LIN {X 0,Y 199.648,Z 315.611,A -85,B 0,C 180,E1 -21577.217,E2 -21577.217} C_VEL
LIN {X 0,Y 199.715,Z 315.609,A -85,B 0,C 180,E1 -21581.799,E2 -21581.799} C_VEL
LIN {X 0,Y 199.766,Z 315.596,A -85,B 0,C 180,E1 -21585.742,E2 -21585.742} C_VEL
LIN {X 0,Y 199.991,Z 315.572,A -85,B 0,C 180,E1 -21589.879,E2 -21589.879} C_VEL
LIN {X 0,Y 199.982,Z 315.569,A -85,B 0,C 180,E1 -21593.947,E2 -21593.947} C_VEL
LIN {X 0,Y 200.285,Z 315.535,A -85,B 0,C 180,E1 -21597.988,E2 -21597.988} C_VEL
LIN {X 0,Y 200.436,Z 315.515,A -85,B 0,C 180,E1 -21599.999,E2 -21599.999} C_VEL
LIN {X 0,Y 199.983,Z 315.57,A -85,B 0,C 180,E1 -21604.029,E2 -21604.029} C_VEL
LIN {X 0,Y 200.046,Z 315.564,A -85,B 0,C 180,E1 -21608.077,E2 -21608.077} C_VEL
LIN {X 0,Y 199.831,Z 315.588,A -85,B 0,C 180,E1 -21612.181,E2 -21612.181} C_VEL
LIN {X 0,Y 199.759,Z 315.601,A -85,B 0,C 180,E1 -21616.346,E2 -21616.346} C_VEL
LIN {X 0,Y 199.644,Z 315.611,A -85,B 0,C 180,E1 -21620.61,E2 -21620.61} C_VEL
LIN {X 0,Y 199.625,Z 315.617,A -85,B 0,C 180,E1 -21624.99,E2 -21624.99} C_VEL
LIN {X 0,Y 199.594,Z 315.616,A -85,B 0,C 180,E1 -21629.534,E2 -21629.534} C_VEL
LIN {X 0,Y 199.635,Z 315.616,A -85,B 0,C 180,E1 -21632.355,E2 -21632.355} C_VEL
LIN {X 0,Y 199.59,Z 315.623,A -85,B 0,C 180,E1 -21636.769,E2 -21636.769} C_VEL
LIN {X 0,Y 199.569,Z 315.628,A -85,B 0,C 180,E1 -21639.336,E2 -21639.336} C_VEL
LIN {X 0,Y 199.544,Z 315.627,A -85,B 0,C 180,E1 -21642.313,E2 -21642.313} C_VEL
LIN {X 0,Y 199.554,Z 315.629,A -85,B 0,C 180,E1 -21645.233,E2 -21645.233} C_VEL
LIN {X 0,Y 199.69,Z 315.812,A -85,B 0,C 180,E1 -21650.538,E2 -21650.538} C_VEL
LIN {X 0,Y 202.068,Z 326.672,A -85,B 0,C 180,E1 -21654.989,E2 -21654.989} C_VEL
LIN {X 0,Y 204.574,Z 338.295,A -85,B 0,C 180,E1 -21659.506,E2 -21659.506} C_VEL
LIN {X 0,Y 205.421,Z 343.365,A -85,B 0,C 180,E1 -21661.389,E2 -21661.389} C_VEL
LIN {X 0,Y 205.397,Z 343.737,A -85,B 0,C 180,E1 -21661.521,E2 -21661.521} C_VEL
LIN {X 0,Y 206.412,Z 366.002,A -85,B 0,C 180,E1 -21662.678,E2 -21662.678} C_VEL
LIN {X 0,Y 207.666,Z 381.182,A -85,B 0,C 180,E1 -21663.491,E2 -21663.491} C_VEL
LIN {X 0,Y 207.515,Z 385.039,A -85,B 0,C 180,E1 -21663.67,E2 -21663.67} C_VEL
LIN {X 0,Y 206.711,Z 388.85,A -85,B 0,C 180,E1 -21663.813,E2 -21663.813} C_VEL
LIN {X 0,Y 200.517,Z 405.605,A -85,B 0,C 180,E1 -21664.357,E2 -21664.357} C_VEL
LIN {X 0,Y 199.538,Z 411.412,A -85,B 0,C 180,E1 -21664.613,E2 -21664.613} C_VEL
LIN {X 0,Y 198.167,Z 444.281,A -85,B 0,C 180,E1 -21666.285,E2 -21666.285} C_VEL
LIN {X 0,Y 197.452,Z 454.911,A -85,B 0,C 180,E1 -21667.096,E2 -21667.096} C_VEL
LIN {X 0,Y 196.39,Z 466.849,A -85,B 0,C 180,E1 -21668.351,E2 -21668.351} C_VEL
LIN {X 0,Y 195.216,Z 478.665,A -85,B 0,C 180,E1 -21670.039,E2 -21670.039} C_VEL
LIN {X 0,Y 194.149,Z 488.366,A -85,B 0,C 180,E1 -21671.813,E2 -21671.813} C_VEL
LIN {X 0,Y 193.082,Z 497.591,A -85,B 0,C 180,E1 -21673.892,E2 -21673.892} C_VEL
LIN {X 0,Y 192.324,Z 504.426,A -85,B 0,C 180,E1 -21675.726,E2 -21675.726} C_VEL
LIN {X 0,Y 191.715,Z 511.1,A -85,B 0,C 180,E1 -21677.837,E2 -21677.837} C_VEL
LIN {X 0,Y 191.271,Z 518.01,A -85,B 0,C 180,E1 -21680.488,E2 -21680.488} C_VEL
LIN {X 0,Y 191.048,Z 523.997,A -85,B 0,C 180,E1 -21683.323,E2 -21683.323} C_VEL
LIN {X 0,Y 190.99,Z 528.22,A -85,B 0,C 180,E1 -21685.784,E2 -21685.784} C_VEL
LIN {X 0,Y 190.988,Z 532.388,A -85,B 0,C 180,E1 -21688.95,E2 -21688.95} C_VEL
LIN {X 0,Y 191.131,Z 533.502,A -85,B 0,C 180,E1 -21690.004,E2 -21690.004} C_VEL
LIN {X 0,Y 190.578,Z 536.736,A -85,B 0,C 180,E1 -21694.234,E2 -21694.234} C_VEL
LIN {X 0,Y 190.558,Z 538.115,A -85,B 0,C 180,E1 -21698.487,E2 -21698.487} C_VEL
LIN {X 0,Y 190.933,Z 538.228,A -85,B 0,C 180,E1 -21700.609,E2 -21700.609} C_VEL
LIN {X 0,Y 192.399,Z 537.275,A -85,B 0,C 180,E1 -21704.818,E2 -21704.818} C_VEL
LIN {X 0,Y 195.192,Z 534.63,A -85,B 0,C 180,E1 -21708.91,E2 -21708.91} C_VEL
LIN {X 0,Y 197.896,Z 531.626,A -85,B 0,C 180,E1 -21711.896,E2 -21711.896} C_VEL
LIN {X 0,Y 201.136,Z 527.628,A -85,B 0,C 180,E1 -21714.792,E2 -21714.792} C_VEL
LIN {X 0,Y 205.16,Z 522.48,A -85,B 0,C 180,E1 -21717.547,E2 -21717.547} C_VEL
LIN {X 0,Y 208.994,Z 517.234,A -85,B 0,C 180,E1 -21719.738,E2 -21719.738} C_VEL
LIN {X 0,Y 213.102,Z 511.034,A -85,B 0,C 180,E1 -21721.849,E2 -21721.849} C_VEL
LIN {X 0,Y 216.699,Z 505.229,A -85,B 0,C 180,E1 -21723.46,E2 -21723.46} C_VEL
LIN {X 0,Y 221.524,Z 496.519,A -85,B 0,C 180,E1 -21725.38,E2 -21725.38} C_VEL
LIN {X 0,Y 225.582,Z 488.226,A -85,B 0,C 180,E1 -21726.851,E2 -21726.851} C_VEL
LIN {X 0,Y 229.297,Z 479.732,A -85,B 0,C 180,E1 -21728.085,E2 -21728.085} C_VEL
LIN {X 0,Y 232.642,Z 471.031,A -85,B 0,C 180,E1 -21729.096,E2 -21729.096} C_VEL
LIN {X 0,Y 236.162,Z 460.215,A -85,B 0,C 180,E1 -21730.056,E2 -21730.056} C_VEL
LIN {X 0,Y 238.892,Z 449.846,A -85,B 0,C 180,E1 -21730.748,E2 -21730.748} C_VEL
LIN {X 0,Y 241.019,Z 439.165,A -85,B 0,C 180,E1 -21731.279,E2 -21731.279} C_VEL
LIN {X 0,Y 246.635,Z 399.578,A -85,B 0,C 180,E1 -21732.928,E2 -21732.928} C_VEL
LIN {X 0,Y 244.463,Z 393.666,A -85,B 0,C 180,E1 -21734.894,E2 -21734.894} C_VEL
LIN {X 0,Y 242.901,Z 389.862,A -85,B 0,C 180,E1 -21736.566,E2 -21736.566} C_VEL
LIN {X 0,Y 241.28,Z 386.207,A -85,B 0,C 180,E1 -21738.592,E2 -21738.592} C_VEL
LIN {X 0,Y 239.343,Z 382.083,A -85,B 0,C 180,E1 -21742.091,E2 -21742.091} C_VEL
LIN {X 0,Y 238.603,Z 380.779,A -85,B 0,C 180,E1 -21744.45,E2 -21744.45} C_VEL
LIN {X 0,Y 238.575,Z 380.682,A -85,B 0,C 180,E1 -21748.678,E2 -21748.678} C_VEL
LIN {X 0,Y 239.448,Z 381.752,A -85,B 0,C 180,E1 -21751.296,E2 -21751.296} C_VEL
LIN {X 0,Y 241.721,Z 386.414,A -85,B 0,C 180,E1 -21755.249,E2 -21755.249} C_VEL
LIN {X 0,Y 243.812,Z 390.848,A -85,B 0,C 180,E1 -21757.643,E2 -21757.643} C_VEL
LIN {X 0,Y 245.743,Z 395.641,A -85,B 0,C 180,E1 -21759.539,E2 -21759.539} C_VEL
LIN {X 0,Y 246.432,Z 397.591,A -85,B 0,C 180,E1 -21760.175,E2 -21760.175} C_VEL
LIN {X 0,Y 240.499,Z 435.091,A -85,B 0,C 180,E1 -21761.871,E2 -21761.871} C_VEL
LIN {X 0,Y 237.483,Z 448.761,A -85,B 0,C 180,E1 -21762.787,E2 -21762.787} C_VEL
LIN {X 0,Y 234.505,Z 458.837,A -85,B 0,C 180,E1 -21763.725,E2 -21763.725} C_VEL
LIN {X 0,Y 231.305,Z 467.899,A -85,B 0,C 180,E1 -21764.808,E2 -21764.808} C_VEL
LIN {X 0,Y 227.57,Z 476.863,A -85,B 0,C 180,E1 -21766.153,E2 -21766.153} C_VEL
LIN {X 0,Y 223.672,Z 484.895,A -85,B 0,C 180,E1 -21767.65,E2 -21767.65} C_VEL
LIN {X 0,Y 219.496,Z 492.508,A -85,B 0,C 180,E1 -21769.392,E2 -21769.392} C_VEL
LIN {X 0,Y 214.975,Z 499.839,A -85,B 0,C 180,E1 -21771.541,E2 -21771.541} C_VEL
LIN {X 0,Y 209.923,Z 506.722,A -85,B 0,C 180,E1 -21774.237,E2 -21774.237} C_VEL
LIN {X 0,Y 205.514,Z 511.853,A -85,B 0,C 180,E1 -21776.975,E2 -21776.975} C_VEL
LIN {X 0,Y 202.853,Z 514.621,A -85,B 0,C 180,E1 -21778.909,E2 -21778.909} C_VEL
LIN {X 0,Y 199.2,Z 517.68,A -85,B 0,C 180,E1 -21782.023,E2 -21782.023} C_VEL
LIN {X 0,Y 197.206,Z 519.017,A -85,B 0,C 180,E1 -21784.088,E2 -21784.088} C_VEL
LIN {X 0,Y 195.451,Z 519.821,A -85,B 0,C 180,E1 -21786.194,E2 -21786.194} C_VEL
LIN {X 0,Y 193.934,Z 520.014,A -85,B 0,C 180,E1 -21788.336,E2 -21788.336} C_VEL
LIN {X 0,Y 192.716,Z 519.734,A -85,B 0,C 180,E1 -21790.507,E2 -21790.507} C_VEL
LIN {X 0,Y 191.73,Z 518.983,A -85,B 0,C 180,E1 -21792.706,E2 -21792.706} C_VEL
LIN {X 0,Y 190.999,Z 517.686,A -85,B 0,C 180,E1 -21794.927,E2 -21794.927} C_VEL
LIN {X 0,Y 190.342,Z 514.593,A -85,B 0,C 180,E1 -21798.292,E2 -21798.292} C_VEL
LIN {X 0,Y 190.255,Z 511.807,A -85,B 0,C 180,E1 -21800.545,E2 -21800.545} C_VEL
LIN {X 0,Y 190.441,Z 506.225,A -85,B 0,C 180,E1 -21803.951,E2 -21803.951} C_VEL
LIN {X 0,Y 190.888,Z 500.472,A -85,B 0,C 180,E1 -21806.689,E2 -21806.689} C_VEL
LIN {X 0,Y 191.39,Z 494.218,A -85,B 0,C 180,E1 -21809.115,E2 -21809.115} C_VEL
LIN {X 0,Y 191.861,Z 488.925,A -85,B 0,C 180,E1 -21810.854,E2 -21810.854} C_VEL
LIN {X 0,Y 192.742,Z 480.468,A -85,B 0,C 180,E1 -21813.159,E2 -21813.159} C_VEL
LIN {X 0,Y 193.68,Z 471.435,A -85,B 0,C 180,E1 -21815.175,E2 -21815.175} C_VEL
LIN {X 0,Y 194.762,Z 460.212,A -85,B 0,C 180,E1 -21817.189,E2 -21817.189} C_VEL
LIN {X 0,Y 195.736,Z 448.504,A -85,B 0,C 180,E1 -21818.765,E2 -21818.765} C_VEL
LIN {X 0,Y 196.492,Z 438.184,A -85,B 0,C 180,E1 -21819.827,E2 -21819.827} C_VEL
LIN {X 0,Y 197.164,Z 426.158,A -85,B 0,C 180,E1 -21820.726,E2 -21820.726} C_VEL
LIN {X 0,Y 199.44,Z 377.415,A -85,B 0,C 180,E1 -21823.388,E2 -21823.388} C_VEL
LIN {X 0,Y 196.403,Z 343.515,A -85,B 0,C 180,E1 -21825.476,E2 -21825.476} C_VEL
LIN {X 0,Y 196.313,Z 340.974,A -85,B 0,C 180,E1 -21825.635,E2 -21825.635} C_VEL
LIN {X 0,Y 196.727,Z 336.975,A -85,B 0,C 180,E1 -21827.252,E2 -21827.252} C_VEL
LIN {X 0,Y 194.607,Z 325.863,A -85,B 0,C 180,E1 -21832.125,E2 -21832.125} C_VEL
LIN {X 0,Y 192.67,Z 316.483,A -85,B 0,C 180,E1 -21836.514,E2 -21836.514} C_VEL
LIN {X 0,Y 192.616,Z 316.492,A -85,B 0,C 180,E1 -21841.682,E2 -21841.682} C_VEL
LIN {X 0,Y 192.662,Z 316.489,A -85,B 0,C 180,E1 -21846.341,E2 -21846.341} C_VEL
LIN {X 0,Y 192.701,Z 316.479,A -85,B 0,C 180,E1 -21851.49,E2 -21851.49} C_VEL
LIN {X 0,Y 192.735,Z 316.472,A -85,B 0,C 180,E1 -21855.209,E2 -21855.209} C_VEL
LIN {X 0,Y 192.952,Z 316.449,A -85,B 0,C 180,E1 -21859.564,E2 -21859.564} C_VEL
LIN {X 0,Y 192.968,Z 316.444,A -85,B 0,C 180,E1 -21863.724,E2 -21863.724} C_VEL
LIN {X 0,Y 193.231,Z 316.415,A -85,B 0,C 180,E1 -21867.912,E2 -21867.912} C_VEL
LIN {X 0,Y 193.417,Z 316.392,A -85,B 0,C 180,E1 -21869.996,E2 -21869.996} C_VEL
LIN {X 0,Y 192.934,Z 316.449,A -85,B 0,C 180,E1 -21874.173,E2 -21874.173} C_VEL
LIN {X 0,Y 193.028,Z 316.441,A -85,B 0,C 180,E1 -21878.369,E2 -21878.369} C_VEL
LIN {X 0,Y 192.794,Z 316.466,A -85,B 0,C 180,E1 -21882.628,E2 -21882.628} C_VEL
LIN {X 0,Y 192.715,Z 316.48,A -85,B 0,C 180,E1 -21886.956,E2 -21886.956} C_VEL
LIN {X 0,Y 192.578,Z 316.491,A -85,B 0,C 180,E1 -21891.397,E2 -21891.397} C_VEL
LIN {X 0,Y 192.63,Z 316.487,A -85,B 0,C 180,E1 -21894.198,E2 -21894.198} C_VEL
LIN {X 0,Y 192.593,Z 316.492,A -85,B 0,C 180,E1 -21898.858,E2 -21898.858} C_VEL
LIN {X 0,Y 192.584,Z 316.493,A -85,B 0,C 180,E1 -21903.18,E2 -21903.18} C_VEL
LIN {X 0,Y 192.528,Z 316.498,A -85,B 0,C 180,E1 -21908.347,E2 -21908.347} C_VEL
LIN {X 0,Y 192.471,Z 316.508,A -85,B 0,C 180,E1 -21913.087,E2 -21913.087} C_VEL
LIN {X 0,Y 192.468,Z 316.506,A -85,B 0,C 180,E1 -21916.9,E2 -21916.9} C_VEL
LIN {X 0,Y 192.52,Z 316.501,A -85,B 0,C 180,E1 -21921.639,E2 -21921.639} C_VEL
LIN {X 0,Y 192.572,Z 316.494,A -85,B 0,C 180,E1 -21926.808,E2 -21926.808} C_VEL
LIN {X 0,Y 192.638,Z 316.488,A -85,B 0,C 180,E1 -21931.686,E2 -21931.686} C_VEL
LIN {X 0,Y 192.644,Z 316.482,A -85,B 0,C 180,E1 -21936.339,E2 -21936.339} C_VEL
LIN {X 0,Y 192.664,Z 316.486,A -85,B 0,C 180,E1 -21941.488,E2 -21941.488} C_VEL
LIN {X 0,Y 192.692,Z 316.475,A -85,B 0,C 180,E1 -21945.207,E2 -21945.207} C_VEL
LIN {X 0,Y 192.914,Z 316.453,A -85,B 0,C 180,E1 -21949.564,E2 -21949.564} C_VEL
LIN {X 0,Y 192.944,Z 316.445,A -85,B 0,C 180,E1 -21953.725,E2 -21953.725} C_VEL
LIN {X 0,Y 193.227,Z 316.414,A -85,B 0,C 180,E1 -21957.914,E2 -21957.914} C_VEL
LIN {X 0,Y 193.401,Z 316.392,A -85,B 0,C 180,E1 -21959.999,E2 -21959.999} C_VEL
LIN {X 0,Y 192.929,Z 316.448,A -85,B 0,C 180,E1 -21964.177,E2 -21964.177} C_VEL
LIN {X 0,Y 192.996,Z 316.442,A -85,B 0,C 180,E1 -21968.374,E2 -21968.374} C_VEL
LIN {X 0,Y 192.759,Z 316.469,A -85,B 0,C 180,E1 -21972.635,E2 -21972.635} C_VEL
LIN {X 0,Y 192.717,Z 316.477,A -85,B 0,C 180,E1 -21976.961,E2 -21976.961} C_VEL
LIN {X 0,Y 192.578,Z 316.491,A -85,B 0,C 180,E1 -21981.403,E2 -21981.403} C_VEL
LIN {X 0,Y 192.61,Z 316.493,A -85,B 0,C 180,E1 -21984.211,E2 -21984.211} C_VEL
LIN {X 0,Y 192.592,Z 316.489,A -85,B 0,C 180,E1 -21988.88,E2 -21988.88} C_VEL
LIN {X 0,Y 192.566,Z 316.498,A -85,B 0,C 180,E1 -21993.191,E2 -21993.191} C_VEL
LIN {X 0,Y 192.516,Z 316.504,A -85,B 0,C 180,E1 -21998.359,E2 -21998.359} C_VEL
LIN {X 0,Y 192.463,Z 316.512,A -85,B 0,C 180,E1 -22003.099,E2 -22003.099} C_VEL
LIN {X 0,Y 192.467,Z 316.51,A -85,B 0,C 180,E1 -22006.911,E2 -22006.911} C_VEL
LIN {X 0,Y 192.604,Z 316.676,A -85,B 0,C 180,E1 -22010.019,E2 -22010.019} C_VEL
LIN {X 0,Y 194.779,Z 326.353,A -85,B 0,C 180,E1 -22014.143,E2 -22014.143} C_VEL
LIN {X 0,Y 197.226,Z 337.828,A -85,B 0,C 180,E1 -22018.782,E2 -22018.782} C_VEL
LIN {X 0,Y 198.356,Z 343.639,A -85,B 0,C 180,E1 -22021.049,E2 -22021.049} C_VEL
LIN {X 0,Y 199.807,Z 370.761,A -85,B 0,C 180,E1 -22022.547,E2 -22022.547} C_VEL
LIN {X 0,Y 200.674,Z 384.052,A -85,B 0,C 180,E1 -22023.276,E2 -22023.276} C_VEL
LIN {X 0,Y 199.538,Z 411.412,A -85,B 0,C 180,E1 -22024.613,E2 -22024.613} C_VEL
LIN {X 0,Y 198.65,Z 417.188,A -85,B 0,C 180,E1 -22024.865,E2 -22024.865} C_VEL
LIN {X 0,Y 192.214,Z 435.809,A -85,B 0,C 180,E1 -22025.563,E2 -22025.563} C_VEL
LIN {X 0,Y 191.277,Z 441.55,A -85,B 0,C 180,E1 -22025.881,E2 -22025.881} C_VEL
LIN {X 0,Y 190.616,Z 452.157,A -85,B 0,C 180,E1 -22026.657,E2 -22026.657} C_VEL
LIN {X 0,Y 189.733,Z 462.427,A -85,B 0,C 180,E1 -22027.695,E2 -22027.695} C_VEL
LIN {X 0,Y 188.828,Z 471.698,A -85,B 0,C 180,E1 -22028.901,E2 -22028.901} C_VEL
LIN {X 0,Y 187.89,Z 480.588,A -85,B 0,C 180,E1 -22030.334,E2 -22030.334} C_VEL
LIN {X 0,Y 186.975,Z 488.81,A -85,B 0,C 180,E1 -22031.941,E2 -22031.941} C_VEL
LIN {X 0,Y 186.029,Z 496.842,A -85,B 0,C 180,E1 -22033.828,E2 -22033.828} C_VEL
LIN {X 0,Y 185.277,Z 503.711,A -85,B 0,C 180,E1 -22035.732,E2 -22035.732} C_VEL
LIN {X 0,Y 184.574,Z 511.846,A -85,B 0,C 180,E1 -22038.474,E2 -22038.474} C_VEL
LIN {X 0,Y 184.224,Z 517.336,A -85,B 0,C 180,E1 -22040.675,E2 -22040.675} C_VEL
LIN {X 0,Y 184.043,Z 523.013,A -85,B 0,C 180,E1 -22043.427,E2 -22043.427} C_VEL
LIN {X 0,Y 183.993,Z 526.802,A -85,B 0,C 180,E1 -22045.624,E2 -22045.624} C_VEL
LIN {X 0,Y 183.975,Z 531.244,A -85,B 0,C 180,E1 -22048.91,E2 -22048.91} C_VEL
LIN {X 0,Y 184.118,Z 532.372,A -85,B 0,C 180,E1 -22050.004,E2 -22050.004} C_VEL
LIN {X 0,Y 183.695,Z 534.391,A -85,B 0,C 180,E1 -22052.197,E2 -22052.197} C_VEL
LIN {X 0,Y 183.455,Z 536.25,A -85,B 0,C 180,E1 -22055.117,E2 -22055.117} C_VEL
LIN {X 0,Y 183.535,Z 537.535,A -85,B 0,C 180,E1 -22058.814,E2 -22058.814} C_VEL
LIN {X 0,Y 184.599,Z 537.553,A -85,B 0,C 180,E1 -22063.208,E2 -22063.208} C_VEL
LIN {X 0,Y 185.515,Z 537.031,A -85,B 0,C 180,E1 -22065.381,E2 -22065.381} C_VEL
LIN {X 0,Y 188.465,Z 534.759,A -85,B 0,C 180,E1 -22069.613,E2 -22069.613} C_VEL
LIN {X 0,Y 191.326,Z 531.999,A -85,B 0,C 180,E1 -22072.689,E2 -22072.689} C_VEL
LIN {X 0,Y 194.746,Z 528.239,A -85,B 0,C 180,E1 -22075.664,E2 -22075.664} C_VEL
LIN {X 0,Y 198.959,Z 523.417,A -85,B 0,C 180,E1 -22078.483,E2 -22078.483} C_VEL
LIN {X 0,Y 203.777,Z 517.353,A -85,B 0,C 180,E1 -22081.155,E2 -22081.155} C_VEL
LIN {X 0,Y 208.14,Z 511.24,A -85,B 0,C 180,E1 -22083.278,E2 -22083.278} C_VEL
LIN {X 0,Y 212.908,Z 503.926,A -85,B 0,C 180,E1 -22085.287,E2 -22085.287} C_VEL
LIN {X 0,Y 216.99,Z 497.107,A -85,B 0,C 180,E1 -22086.812,E2 -22086.812} C_VEL
LIN {X 0,Y 221.791,Z 487.937,A -85,B 0,C 180,E1 -22088.453,E2 -22088.453} C_VEL
LIN {X 0,Y 225.676,Z 479.438,A -85,B 0,C 180,E1 -22089.673,E2 -22089.673} C_VEL
LIN {X 0,Y 229.172,Z 470.724,A -85,B 0,C 180,E1 -22090.667,E2 -22090.667} C_VEL
LIN {X 0,Y 232.839,Z 460.044,A -85,B 0,C 180,E1 -22091.609,E2 -22091.609} C_VEL
LIN {X 0,Y 235.699,Z 449.867,A -85,B 0,C 180,E1 -22092.28,E2 -22092.28} C_VEL
LIN {X 0,Y 238.021,Z 438.815,A -85,B 0,C 180,E1 -22092.842,E2 -22092.842} C_VEL
LIN {X 0,Y 243.371,Z 403.423,A -85,B 0,C 180,E1 -22094.277,E2 -22094.277} C_VEL
LIN {X 0,Y 241.701,Z 398.475,A -85,B 0,C 180,E1 -22096.088,E2 -22096.088} C_VEL
LIN {X 0,Y 240.167,Z 394.667,A -85,B 0,C 180,E1 -22097.922,E2 -22097.922} C_VEL
LIN {X 0,Y 239.212,Z 392.39,A -85,B 0,C 180,E1 -22099.353,E2 -22099.353} C_VEL
LIN {X 0,Y 237.653,Z 388.741,A -85,B 0,C 180,E1 -22102.588,E2 -22102.588} C_VEL
LIN {X 0,Y 237.101,Z 387.701,A -85,B 0,C 180,E1 -22104.584,E2 -22104.584} C_VEL
LIN {X 0,Y 237.055,Z 387.575,A -85,B 0,C 180,E1 -22108.467,E2 -22108.467} C_VEL
LIN {X 0,Y 237.83,Z 388.654,A -85,B 0,C 180,E1 -22111.082,E2 -22111.082} C_VEL
LIN {X 0,Y 239.727,Z 392.787,A -85,B 0,C 180,E1 -22114.678,E2 -22114.678} C_VEL
LIN {X 0,Y 241.672,Z 397.356,A -85,B 0,C 180,E1 -22117.164,E2 -22117.164} C_VEL
LIN {X 0,Y 243.093,Z 401.381,A -85,B 0,C 180,E1 -22118.779,E2 -22118.779} C_VEL
LIN {X 0,Y 237.399,Z 436.213,A -85,B 0,C 180,E1 -22120.368,E2 -22120.368} C_VEL
LIN {X 0,Y 234.141,Z 449.81,A -85,B 0,C 180,E1 -22121.29,E2 -22121.29} C_VEL
LIN {X 0,Y 230.829,Z 460.19,A -85,B 0,C 180,E1 -22122.275,E2 -22122.275} C_VEL
LIN {X 0,Y 227.356,Z 469.255,A -85,B 0,C 180,E1 -22123.383,E2 -22123.383} C_VEL
LIN {X 0,Y 223.936,Z 477.009,A -85,B 0,C 180,E1 -22124.529,E2 -22124.529} C_VEL
LIN {X 0,Y 220.707,Z 483.562,A -85,B 0,C 180,E1 -22125.714,E2 -22125.714} C_VEL
LIN {X 0,Y 215.897,Z 491.926,A -85,B 0,C 180,E1 -22127.566,E2 -22127.566} C_VEL
LIN {X 0,Y 211.51,Z 498.627,A -85,B 0,C 180,E1 -22129.471,E2 -22129.471} C_VEL
LIN {X 0,Y 206.908,Z 504.866,A -85,B 0,C 180,E1 -22131.701,E2 -22131.701} C_VEL
LIN {X 0,Y 202.663,Z 509.87,A -85,B 0,C 180,E1 -22134.03,E2 -22134.03} C_VEL
LIN {X 0,Y 198.198,Z 514.369,A -85,B 0,C 180,E1 -22136.85,E2 -22136.85} C_VEL
LIN {X 0,Y 194.112,Z 517.698,A -85,B 0,C 180,E1 -22140.001,E2 -22140.001} C_VEL
LIN {X 0,Y 191.8,Z 519.195,A -85,B 0,C 180,E1 -22142.101,E2 -22142.101} C_VEL
LIN {X 0,Y 189.781,Z 520.062,A -85,B 0,C 180,E1 -22144.249,E2 -22144.249} C_VEL
LIN {X 0,Y 188.012,Z 520.468,A -85,B 0,C 180,E1 -22146.44,E2 -22146.44} C_VEL
LIN {X 0,Y 186.554,Z 520.424,A -85,B 0,C 180,E1 -22148.668,E2 -22148.668} C_VEL
LIN {X 0,Y 185.338,Z 519.826,A -85,B 0,C 180,E1 -22150.931,E2 -22150.931} C_VEL
LIN {X 0,Y 184.412,Z 518.619,A -85,B 0,C 180,E1 -22153.22,E2 -22153.22} C_VEL
LIN {X 0,Y 183.48,Z 515.864,A -85,B 0,C 180,E1 -22156.749,E2 -22156.749} C_VEL
LIN {X 0,Y 183.165,Z 511.873,A -85,B 0,C 180,E1 -22160.203,E2 -22160.203} C_VEL
LIN {X 0,Y 183.282,Z 507.471,A -85,B 0,C 180,E1 -22163.034,E2 -22163.034} C_VEL
LIN {X 0,Y 183.69,Z 501.373,A -85,B 0,C 180,E1 -22166.105,E2 -22166.105} C_VEL
LIN {X 0,Y 184.197,Z 495.138,A -85,B 0,C 180,E1 -22168.652,E2 -22168.652} C_VEL
LIN {X 0,Y 184.799,Z 488.543,A -85,B 0,C 180,E1 -22170.893,E2 -22170.893} C_VEL
LIN {X 0,Y 185.603,Z 480.789,A -85,B 0,C 180,E1 -22173.087,E2 -22173.087} C_VEL
LIN {X 0,Y 186.466,Z 472.258,A -85,B 0,C 180,E1 -22175.086,E2 -22175.086} C_VEL
LIN {X 0,Y 187.578,Z 461.62,A -85,B 0,C 180,E1 -22177.109,E2 -22177.109} C_VEL
LIN {X 0,Y 188.574,Z 449.793,A -85,B 0,C 180,E1 -22178.812,E2 -22178.812} C_VEL
LIN {X 0,Y 189.408,Z 439.144,A -85,B 0,C 180,E1 -22179.971,E2 -22179.971} C_VEL
LIN {X 0,Y 190.024,Z 428.037,A -85,B 0,C 180,E1 -22180.858,E2 -22180.858} C_VEL
LIN {X 0,Y 192.42,Z 377.461,A -85,B 0,C 180,E1 -22183.751,E2 -22183.751} C_VEL
LIN {X 0,Y 189.509,Z 344.606,A -85,B 0,C 180,E1 -22185.853,E2 -22185.853} C_VEL
LIN {X 0,Y 189.385,Z 340.94,A -85,B 0,C 180,E1 -22186.126,E2 -22186.126} C_VEL
LIN {X 0,Y 189.686,Z 337.773,A -85,B 0,C 180,E1 -22187.456,E2 -22187.456} C_VEL
LIN {X 0,Y 187.56,Z 326.77,A -85,B 0,C 180,E1 -22192.448,E2 -22192.448} C_VEL
LIN {X 0,Y 185.62,Z 317.361,A -85,B 0,C 180,E1 -22196.992,E2 -22196.992} C_VEL
LIN {X 0,Y 185.527,Z 317.375,A -85,B 0,C 180,E1 -22200.609,E2 -22200.609} C_VEL
LIN {X 0,Y 185.551,Z 317.371,A -85,B 0,C 180,E1 -22205.375,E2 -22205.375} C_VEL
LIN {X 0,Y 185.632,Z 317.361,A -85,B 0,C 180,E1 -22211.177,E2 -22211.177} C_VEL
LIN {X 0,Y 185.666,Z 317.357,A -85,B 0,C 180,E1 -22214.632,E2 -22214.632} C_VEL
LIN {X 0,Y 185.894,Z 317.329,A -85,B 0,C 180,E1 -22219.416,E2 -22219.416} C_VEL
LIN {X 0,Y 185.933,Z 317.321,A -85,B 0,C 180,E1 -22223.485,E2 -22223.485} C_VEL
LIN {X 0,Y 186.177,Z 317.294,A -85,B 0,C 180,E1 -22227.832,E2 -22227.832} C_VEL
LIN {X 0,Y 186.383,Z 317.268,A -85,B 0,C 180,E1 -22229.996,E2 -22229.996} C_VEL
LIN {X 0,Y 185.883,Z 317.327,A -85,B 0,C 180,E1 -22234.332,E2 -22234.332} C_VEL
LIN {X 0,Y 185.977,Z 317.318,A -85,B 0,C 180,E1 -22238.689,E2 -22238.689} C_VEL
LIN {X 0,Y 185.719,Z 317.346,A -85,B 0,C 180,E1 -22243.118,E2 -22243.118} C_VEL
LIN {X 0,Y 185.651,Z 317.358,A -85,B 0,C 180,E1 -22247.622,E2 -22247.622} C_VEL
LIN {X 0,Y 185.549,Z 317.366,A -85,B 0,C 180,E1 -22252.25,E2 -22252.25} C_VEL
LIN {X 0,Y 185.572,Z 317.367,A -85,B 0,C 180,E1 -22254.639,E2 -22254.639} C_VEL
LIN {X 0,Y 185.535,Z 317.37,A -85,B 0,C 180,E1 -22259.492,E2 -22259.492} C_VEL
LIN {X 0,Y 185.486,Z 317.378,A -85,B 0,C 180,E1 -22264.626,E2 -22264.626} C_VEL
LIN {X 0,Y 185.487,Z 317.378,A -85,B 0,C 180,E1 -22267.308,E2 -22267.308} C_VEL
LIN {X 0,Y 185.448,Z 317.381,A -85,B 0,C 180,E1 -22270.715,E2 -22270.715} C_VEL
LIN {X 0,Y 185.439,Z 317.385,A -85,B 0,C 180,E1 -22276.049,E2 -22276.049} C_VEL
LIN {X 0,Y 185.436,Z 317.382,A -85,B 0,C 180,E1 -22279.886,E2 -22279.886} C_VEL
LIN {X 0,Y 185.479,Z 317.382,A -85,B 0,C 180,E1 -22282.708,E2 -22282.708} C_VEL
LIN {X 0,Y 185.518,Z 317.37,A -85,B 0,C 180,E1 -22287.969,E2 -22287.969} C_VEL
LIN {X 0,Y 185.557,Z 317.369,A -85,B 0,C 180,E1 -22290.571,E2 -22290.571} C_VEL
LIN {X 0,Y 185.554,Z 317.368,A -85,B 0,C 180,E1 -22295.376,E2 -22295.376} C_VEL
LIN {X 0,Y 185.595,Z 317.365,A -85,B 0,C 180,E1 -22301.176,E2 -22301.176} C_VEL
LIN {X 0,Y 185.677,Z 317.353,A -85,B 0,C 180,E1 -22306.872,E2 -22306.872} C_VEL
LIN {X 0,Y 185.942,Z 317.32,A -85,B 0,C 180,E1 -22311.303,E2 -22311.303} C_VEL
LIN {X 0,Y 186.171,Z 317.293,A -85,B 0,C 180,E1 -22317.835,E2 -22317.835} C_VEL
LIN {X 0,Y 186.365,Z 317.268,A -85,B 0,C 180,E1 -22319.999,E2 -22319.999} C_VEL
LIN {X 0,Y 185.876,Z 317.327,A -85,B 0,C 180,E1 -22324.336,E2 -22324.336} C_VEL
LIN {X 0,Y 185.944,Z 317.321,A -85,B 0,C 180,E1 -22328.694,E2 -22328.694} C_VEL
LIN {X 0,Y 185.687,Z 317.35,A -85,B 0,C 180,E1 -22333.125,E2 -22333.125} C_VEL
LIN {X 0,Y 185.653,Z 317.359,A -85,B 0,C 180,E1 -22337.627,E2 -22337.627} C_VEL
LIN {X 0,Y 185.54,Z 317.372,A -85,B 0,C 180,E1 -22342.257,E2 -22342.257} C_VEL
LIN {X 0,Y 185.495,Z 317.376,A -85,B 0,C 180,E1 -22347.041,E2 -22347.041} C_VEL
LIN {X 0,Y 185.52,Z 317.368,A -85,B 0,C 180,E1 -22349.502,E2 -22349.502} C_VEL
LIN {X 0,Y 185.469,Z 317.383,A -85,B 0,C 180,E1 -22354.637,E2 -22354.637} C_VEL
LIN {X 0,Y 185.474,Z 317.383,A -85,B 0,C 180,E1 -22357.319,E2 -22357.319} C_VEL
LIN {X 0,Y 185.438,Z 317.387,A -85,B 0,C 180,E1 -22360.726,E2 -22360.726} C_VEL
LIN {X 0,Y 185.436,Z 317.386,A -85,B 0,C 180,E1 -22366.061,E2 -22366.061} C_VEL
LIN {X 0,Y 185.555,Z 317.577,A -85,B 0,C 180,E1 -22369.49,E2 -22369.49} C_VEL
LIN {X 0,Y 187.691,Z 327.13,A -85,B 0,C 180,E1 -22373.728,E2 -22373.728} C_VEL
LIN {X 0,Y 190.332,Z 339.442,A -85,B 0,C 180,E1 -22378.881,E2 -22378.881} C_VEL
LIN {X 0,Y 191.25,Z 343.889,A -85,B 0,C 180,E1 -22380.612,E2 -22380.612} C_VEL
LIN {X 0,Y 191.623,Z 350.087,A -85,B 0,C 180,E1 -22380.971,E2 -22380.971} C_VEL
LIN {X 0,Y 193.318,Z 377.402,A -85,B 0,C 180,E1 -22382.541,E2 -22382.541} C_VEL
LIN {X 0,Y 193.719,Z 383.613,A -85,B 0,C 180,E1 -22382.894,E2 -22382.894} C_VEL
LIN {X 0,Y 191.277,Z 441.55,A -85,B 0,C 180,E1 -22385.881,E2 -22385.881} C_VEL
LIN {X 0,Y 190.704,Z 445.375,A -85,B 0,C 180,E1 -22386.111,E2 -22386.111} C_VEL
LIN {X 0,Y 188.208,Z 452.712,A -85,B 0,C 180,E1 -22386.622,E2 -22386.622} C_VEL
LIN {X 0,Y 182.987,Z 464.981,A -85,B 0,C 180,E1 -22387.87,E2 -22387.87} C_VEL
LIN {X 0,Y 181.85,Z 470.285,A -85,B 0,C 180,E1 -22388.621,E2 -22388.621} C_VEL
LIN {X 0,Y 180.912,Z 479.462,A -85,B 0,C 180,E1 -22390.135,E2 -22390.135} C_VEL
LIN {X 0,Y 179.812,Z 488.993,A -85,B 0,C 180,E1 -22392.08,E2 -22392.08} C_VEL
LIN {X 0,Y 178.907,Z 496.948,A -85,B 0,C 180,E1 -22394.045,E2 -22394.045} C_VEL
LIN {X 0,Y 178.075,Z 504.588,A -85,B 0,C 180,E1 -22396.308,E2 -22396.308} C_VEL
LIN {X 0,Y 177.531,Z 511.081,A -85,B 0,C 180,E1 -22398.59,E2 -22398.59} C_VEL
LIN {X 0,Y 177.15,Z 517.934,A -85,B 0,C 180,E1 -22401.507,E2 -22401.507} C_VEL
LIN {X 0,Y 177.027,Z 522.574,A -85,B 0,C 180,E1 -22403.865,E2 -22403.865} C_VEL
LIN {X 0,Y 176.953,Z 526.989,A -85,B 0,C 180,E1 -22406.59,E2 -22406.59} C_VEL
LIN {X 0,Y 177.105,Z 531.229,A -85,B 0,C 180,E1 -22410.005,E2 -22410.005} C_VEL
LIN {X 0,Y 176.695,Z 533.28,A -85,B 0,C 180,E1 -22412.284,E2 -22412.284} C_VEL
LIN {X 0,Y 176.439,Z 535.241,A -85,B 0,C 180,E1 -22415.257,E2 -22415.257} C_VEL
LIN {X 0,Y 176.531,Z 536.796,A -85,B 0,C 180,E1 -22419.167,E2 -22419.167} C_VEL
LIN {X 0,Y 177.669,Z 537.201,A -85,B 0,C 180,E1 -22423.733,E2 -22423.733} C_VEL
LIN {X 0,Y 180.089,Z 535.938,A -85,B 0,C 180,E1 -22428.195,E2 -22428.195} C_VEL
LIN {X 0,Y 181.765,Z 534.799,A -85,B 0,C 180,E1 -22430.367,E2 -22430.367} C_VEL
LIN {X 0,Y 185.942,Z 531.193,A -85,B 0,C 180,E1 -22434.57,E2 -22434.57} C_VEL
LIN {X 0,Y 189.852,Z 527.391,A -85,B 0,C 180,E1 -22437.565,E2 -22437.565} C_VEL
LIN {X 0,Y 194.364,Z 522.49,A -85,B 0,C 180,E1 -22440.414,E2 -22440.414} C_VEL
LIN {X 0,Y 199.544,Z 516.353,A -85,B 0,C 180,E1 -22443.088,E2 -22443.088} C_VEL
LIN {X 0,Y 204.292,Z 510.201,A -85,B 0,C 180,E1 -22445.187,E2 -22445.187} C_VEL
LIN {X 0,Y 209.383,Z 502.822,A -85,B 0,C 180,E1 -22447.17,E2 -22447.17} C_VEL
LIN {X 0,Y 213.676,Z 495.864,A -85,B 0,C 180,E1 -22448.677,E2 -22448.677} C_VEL
LIN {X 0,Y 218.758,Z 486.586,A -85,B 0,C 180,E1 -22450.282,E2 -22450.282} C_VEL
LIN {X 0,Y 222.873,Z 478.011,A -85,B 0,C 180,E1 -22451.468,E2 -22451.468} C_VEL
LIN {X 0,Y 226.549,Z 469.199,A -85,B 0,C 180,E1 -22452.433,E2 -22452.433} C_VEL
LIN {X 0,Y 230.078,Z 459.248,A -85,B 0,C 180,E1 -22453.265,E2 -22453.265} C_VEL
LIN {X 0,Y 233.027,Z 448.965,A -85,B 0,C 180,E1 -22453.921,E2 -22453.921} C_VEL
LIN {X 0,Y 235.439,Z 437.602,A -85,B 0,C 180,E1 -22454.485,E2 -22454.485} C_VEL
LIN {X 0,Y 240.294,Z 407.203,A -85,B 0,C 180,E1 -22455.741,E2 -22455.741} C_VEL
LIN {X 0,Y 238.726,Z 402.587,A -85,B 0,C 180,E1 -22457.682,E2 -22457.682} C_VEL
LIN {X 0,Y 237.5,Z 399.198,A -85,B 0,C 180,E1 -22459.636,E2 -22459.636} C_VEL
LIN {X 0,Y 235.97,Z 395.396,A -85,B 0,C 180,E1 -22463.106,E2 -22463.106} C_VEL
LIN {X 0,Y 235.671,Z 394.712,A -85,B 0,C 180,E1 -22464.336,E2 -22464.336} C_VEL
LIN {X 0,Y 235.414,Z 394.478,A -85,B 0,C 180,E1 -22467.496,E2 -22467.496} C_VEL
LIN {X 0,Y 236.078,Z 395.174,A -85,B 0,C 180,E1 -22470.439,E2 -22470.439} C_VEL
LIN {X 0,Y 237.758,Z 399.147,A -85,B 0,C 180,E1 -22474.097,E2 -22474.097} C_VEL
LIN {X 0,Y 239.335,Z 403.351,A -85,B 0,C 180,E1 -22476.435,E2 -22476.435} C_VEL
LIN {X 0,Y 240.093,Z 405.53,A -85,B 0,C 180,E1 -22477.377,E2 -22477.377} C_VEL
LIN {X 0,Y 234.704,Z 436.401,A -85,B 0,C 180,E1 -22478.767,E2 -22478.767} C_VEL
LIN {X 0,Y 231.358,Z 449.836,A -85,B 0,C 180,E1 -22479.669,E2 -22479.669} C_VEL
LIN {X 0,Y 227.844,Z 460.424,A -85,B 0,C 180,E1 -22480.636,E2 -22480.636} C_VEL
LIN {X 0,Y 224.205,Z 469.581,A -85,B 0,C 180,E1 -22481.733,E2 -22481.733} C_VEL
LIN {X 0,Y 220.14,Z 478.179,A -85,B 0,C 180,E1 -22483.006,E2 -22483.006} C_VEL
LIN {X 0,Y 216.02,Z 485.782,A -85,B 0,C 180,E1 -22484.432,E2 -22484.432} C_VEL
LIN {X 0,Y 210.511,Z 494.635,A -85,B 0,C 180,E1 -22486.486,E2 -22486.486} C_VEL
LIN {X 0,Y 204.383,Z 502.901,A -85,B 0,C 180,E1 -22489.099,E2 -22489.099} C_VEL
LIN {X 0,Y 200.611,Z 507.373,A -85,B 0,C 180,E1 -22490.931,E2 -22490.931} C_VEL
LIN {X 0,Y 195.319,Z 512.683,A -85,B 0,C 180,E1 -22493.804,E2 -22493.804} C_VEL
LIN {X 0,Y 192.156,Z 515.498,A -85,B 0,C 180,E1 -22495.806,E2 -22495.806} C_VEL
LIN {X 0,Y 189.273,Z 517.696,A -85,B 0,C 180,E1 -22497.873,E2 -22497.873} C_VEL
LIN {X 0,Y 186.685,Z 519.236,A -85,B 0,C 180,E1 -22500.001,E2 -22500.001} C_VEL
LIN {X 0,Y 183.077,Z 520.8,A -85,B 0,C 180,E1 -22503.56,E2 -22503.56} C_VEL
LIN {X 0,Y 180.592,Z 521.028,A -85,B 0,C 180,E1 -22506.706,E2 -22506.706} C_VEL
LIN {X 0,Y 178.515,Z 520.171,A -85,B 0,C 180,E1 -22510.195,E2 -22510.195} C_VEL
LIN {X 0,Y 177.081,Z 518.084,A -85,B 0,C 180,E1 -22513.777,E2 -22513.777} C_VEL
LIN {X 0,Y 176.362,Z 515.206,A -85,B 0,C 180,E1 -22516.985,E2 -22516.985} C_VEL
LIN {X 0,Y 176.099,Z 511.815,A -85,B 0,C 180,E1 -22519.831,E2 -22519.831} C_VEL
LIN {X 0,Y 176.193,Z 507.134,A -85,B 0,C 180,E1 -22522.888,E2 -22522.888} C_VEL
LIN {X 0,Y 176.601,Z 501.187,A -85,B 0,C 180,E1 -22525.962,E2 -22525.962} C_VEL
LIN {X 0,Y 177.086,Z 495.284,A -85,B 0,C 180,E1 -22528.442,E2 -22528.442} C_VEL
LIN {X 0,Y 177.739,Z 488.126,A -85,B 0,C 180,E1 -22530.934,E2 -22530.934} C_VEL
LIN {X 0,Y 178.503,Z 480.602,A -85,B 0,C 180,E1 -22533.114,E2 -22533.114} C_VEL
LIN {X 0,Y 179.346,Z 472.34,A -85,B 0,C 180,E1 -22535.107,E2 -22535.107} C_VEL
LIN {X 0,Y 180.411,Z 462.018,A -85,B 0,C 180,E1 -22537.145,E2 -22537.145} C_VEL
LIN {X 0,Y 181.425,Z 450.487,A -85,B 0,C 180,E1 -22538.896,E2 -22538.896} C_VEL
LIN {X 0,Y 182.297,Z 440.552,A -85,B 0,C 180,E1 -22540.05,E2 -22540.05} C_VEL
LIN {X 0,Y 182.899,Z 430.007,A -85,B 0,C 180,E1 -22540.97,E2 -22540.97} C_VEL
LIN {X 0,Y 185.415,Z 377.772,A -85,B 0,C 180,E1 -22544.126,E2 -22544.126} C_VEL
LIN {X 0,Y 182.538,Z 344.592,A -85,B 0,C 180,E1 -22546.322,E2 -22546.322} C_VEL
LIN {X 0,Y 182.47,Z 340.928,A -85,B 0,C 180,E1 -22546.621,E2 -22546.621} C_VEL
LIN {X 0,Y 182.674,Z 338.789,A -85,B 0,C 180,E1 -22547.549,E2 -22547.549} C_VEL
LIN {X 0,Y 180.458,Z 327.498,A -85,B 0,C 180,E1 -22552.867,E2 -22552.867} C_VEL
LIN {X 0,Y 178.532,Z 318.245,A -85,B 0,C 180,E1 -22557.479,E2 -22557.479} C_VEL
LIN {X 0,Y 178.428,Z 318.26,A -85,B 0,C 180,E1 -22561.791,E2 -22561.791} C_VEL
LIN {X 0,Y 178.47,Z 318.255,A -85,B 0,C 180,E1 -22566.807,E2 -22566.807} C_VEL
LIN {X 0,Y 178.613,Z 318.234,A -85,B 0,C 180,E1 -22571.65,E2 -22571.65} C_VEL
LIN {X 0,Y 178.644,Z 318.226,A -85,B 0,C 180,E1 -22576.344,E2 -22576.344} C_VEL
LIN {X 0,Y 178.91,Z 318.199,A -85,B 0,C 180,E1 -22580.956,E2 -22580.956} C_VEL
LIN {X 0,Y 179.125,Z 318.173,A -85,B 0,C 180,E1 -22587.747,E2 -22587.747} C_VEL
LIN {X 0,Y 179.348,Z 318.144,A -85,B 0,C 180,E1 -22589.995,E2 -22589.995} C_VEL
LIN {X 0,Y 178.832,Z 318.205,A -85,B 0,C 180,E1 -22594.503,E2 -22594.503} C_VEL
LIN {X 0,Y 178.907,Z 318.198,A -85,B 0,C 180,E1 -22599.035,E2 -22599.035} C_VEL
LIN {X 0,Y 178.645,Z 318.226,A -85,B 0,C 180,E1 -22603.647,E2 -22603.647} C_VEL
LIN {X 0,Y 178.551,Z 318.242,A -85,B 0,C 180,E1 -22609.145,E2 -22609.145} C_VEL
LIN {X 0,Y 178.51,Z 318.249,A -85,B 0,C 180,E1 -22615.104,E2 -22615.104} C_VEL
LIN {X 0,Y 178.451,Z 318.249,A -85,B 0,C 180,E1 -22620.787,E2 -22620.787} C_VEL
LIN {X 0,Y 178.471,Z 318.253,A -85,B 0,C 180,E1 -22624.211,E2 -22624.211} C_VEL
LIN {X 0,Y 178.374,Z 318.26,A -85,B 0,C 180,E1 -22629.069,E2 -22629.069} C_VEL
LIN {X 0,Y 178.379,Z 318.264,A -85,B 0,C 180,E1 -22632.039,E2 -22632.039} C_VEL
LIN {X 0,Y 178.375,Z 318.264,A -85,B 0,C 180,E1 -22635.158,E2 -22635.158} C_VEL
LIN {X 0,Y 178.379,Z 318.261,A -85,B 0,C 180,E1 -22638.455,E2 -22638.455} C_VEL
LIN {X 0,Y 178.397,Z 318.261,A -85,B 0,C 180,E1 -22643.776,E2 -22643.776} C_VEL
LIN {X 0,Y 178.462,Z 318.252,A -85,B 0,C 180,E1 -22646.54,E2 -22646.54} C_VEL
LIN {X 0,Y 178.498,Z 318.248,A -85,B 0,C 180,E1 -22650.001,E2 -22650.001} C_VEL
LIN {X 0,Y 178.494,Z 318.248,A -85,B 0,C 180,E1 -22654.881,E2 -22654.881} C_VEL
LIN {X 0,Y 178.576,Z 318.241,A -85,B 0,C 180,E1 -22661.647,E2 -22661.647} C_VEL
LIN {X 0,Y 178.604,Z 318.235,A -85,B 0,C 180,E1 -22666.342,E2 -22666.342} C_VEL
LIN {X 0,Y 178.873,Z 318.202,A -85,B 0,C 180,E1 -22670.957,E2 -22670.957} C_VEL
LIN {X 0,Y 179.116,Z 318.172,A -85,B 0,C 180,E1 -22677.75,E2 -22677.75} C_VEL
LIN {X 0,Y 179.329,Z 318.145,A -85,B 0,C 180,E1 -22679.999,E2 -22679.999} C_VEL
LIN {X 0,Y 178.823,Z 318.206,A -85,B 0,C 180,E1 -22684.507,E2 -22684.507} C_VEL
LIN {X 0,Y 178.874,Z 318.203,A -85,B 0,C 180,E1 -22689.041,E2 -22689.041} C_VEL
LIN {X 0,Y 178.616,Z 318.234,A -85,B 0,C 180,E1 -22693.654,E2 -22693.654} C_VEL
LIN {X 0,Y 178.589,Z 318.235,A -85,B 0,C 180,E1 -22699.214,E2 -22699.214} C_VEL
LIN {X 0,Y 178.488,Z 318.25,A -85,B 0,C 180,E1 -22705.115,E2 -22705.115} C_VEL
LIN {X 0,Y 178.434,Z 318.256,A -85,B 0,C 180,E1 -22710.798,E2 -22710.798} C_VEL
LIN {X 0,Y 178.455,Z 318.255,A -85,B 0,C 180,E1 -22714.221,E2 -22714.221} C_VEL
LIN {X 0,Y 178.362,Z 318.27,A -85,B 0,C 180,E1 -22719.082,E2 -22719.082} C_VEL
LIN {X 0,Y 178.37,Z 318.265,A -85,B 0,C 180,E1 -22722.052,E2 -22722.052} C_VEL
LIN {X 0,Y 178.37,Z 318.267,A -85,B 0,C 180,E1 -22725.17,E2 -22725.17} C_VEL
LIN {X 0,Y 178.443,Z 318.316,A -85,B 0,C 180,E1 -22728.87,E2 -22728.87} C_VEL
LIN {X 0,Y 180.436,Z 327.048,A -85,B 0,C 180,E1 -22732.918,E2 -22732.918} C_VEL
LIN {X 0,Y 182.928,Z 338.789,A -85,B 0,C 180,E1 -22738.055,E2 -22738.055} C_VEL
LIN {X 0,Y 183.927,Z 343.642,A -85,B 0,C 180,E1 -22740.1,E2 -22740.1} C_VEL
LIN {X 0,Y 184.6,Z 347.133,A -85,B 0,C 180,E1 -22740.343,E2 -22740.343} C_VEL
LIN {X 0,Y 185.975,Z 372.917,A -85,B 0,C 180,E1 -22741.87,E2 -22741.87} C_VEL
LIN {X 0,Y 186.74,Z 383.572,A -85,B 0,C 180,E1 -22742.504,E2 -22742.504} C_VEL
LIN {X 0,Y 184.194,Z 442.086,A -85,B 0,C 180,E1 -22745.687,E2 -22745.687} C_VEL
LIN {X 0,Y 183.537,Z 452.298,A -85,B 0,C 180,E1 -22746.487,E2 -22746.487} C_VEL
LIN {X 0,Y 182.663,Z 462.218,A -85,B 0,C 180,E1 -22747.543,E2 -22747.543} C_VEL
LIN {X 0,Y 181.85,Z 470.285,A -85,B 0,C 180,E1 -22748.621,E2 -22748.621} C_VEL
LIN {X 0,Y 181.135,Z 473.77,A -85,B 0,C 180,E1 -22749.154,E2 -22749.154} C_VEL
LIN {X 0,Y 178.456,Z 480.349,A -85,B 0,C 180,E1 -22750.28,E2 -22750.28} C_VEL
LIN {X 0,Y 173.06,Z 491.025,A -85,B 0,C 180,E1 -22752.617,E2 -22752.617} C_VEL
LIN {X 0,Y 171.933,Z 495.533,A -85,B 0,C 180,E1 -22753.842,E2 -22753.842} C_VEL
LIN {X 0,Y 171.026,Z 503.75,A -85,B 0,C 180,E1 -22756.339,E2 -22756.339} C_VEL
LIN {X 0,Y 170.5,Z 510.32,A -85,B 0,C 180,E1 -22758.715,E2 -22758.715} C_VEL
LIN {X 0,Y 170.139,Z 517.318,A -85,B 0,C 180,E1 -22761.813,E2 -22761.813} C_VEL
LIN {X 0,Y 170.017,Z 522.286,A -85,B 0,C 180,E1 -22764.472,E2 -22764.472} C_VEL
LIN {X 0,Y 169.989,Z 527.038,A -85,B 0,C 180,E1 -22767.636,E2 -22767.636} C_VEL
LIN {X 0,Y 170.092,Z 529.946,A -85,B 0,C 180,E1 -22770.005,E2 -22770.005} C_VEL
LIN {X 0,Y 169.49,Z 533.864,A -85,B 0,C 180,E1 -22774.761,E2 -22774.761} C_VEL
LIN {X 0,Y 169.329,Z 535.207,A -85,B 0,C 180,E1 -22777.157,E2 -22777.157} C_VEL
LIN {X 0,Y 170,Z 536.586,A -85,B 0,C 180,E1 -22781.933,E2 -22781.933} C_VEL
LIN {X 0,Y 171.825,Z 536.387,A -85,B 0,C 180,E1 -22786.641,E2 -22786.641} C_VEL
LIN {X 0,Y 173.345,Z 535.828,A -85,B 0,C 180,E1 -22788.929,E2 -22788.929} C_VEL
LIN {X 0,Y 177.188,Z 533.322,A -85,B 0,C 180,E1 -22793.371,E2 -22793.371} C_VEL
LIN {X 0,Y 180.954,Z 530.269,A -85,B 0,C 180,E1 -22796.714,E2 -22796.714} C_VEL
LIN {X 0,Y 185.104,Z 526.565,A -85,B 0,C 180,E1 -22799.578,E2 -22799.578} C_VEL
LIN {X 0,Y 190.125,Z 521.636,A -85,B 0,C 180,E1 -22802.413,E2 -22802.413} C_VEL
LIN {X 0,Y 194.706,Z 516.627,A -85,B 0,C 180,E1 -22804.647,E2 -22804.647} C_VEL
LIN {X 0,Y 199.674,Z 510.605,A -85,B 0,C 180,E1 -22806.753,E2 -22806.753} C_VEL
LIN {X 0,Y 205.024,Z 503.431,A -85,B 0,C 180,E1 -22808.726,E2 -22808.726} C_VEL
LIN {X 0,Y 210.646,Z 494.851,A -85,B 0,C 180,E1 -22810.587,E2 -22810.587} C_VEL
LIN {X 0,Y 215.396,Z 486.631,A -85,B 0,C 180,E1 -22811.981,E2 -22811.981} C_VEL
LIN {X 0,Y 219.678,Z 478.11,A -85,B 0,C 180,E1 -22813.144,E2 -22813.144} C_VEL
LIN {X 0,Y 223.524,Z 469.406,A -85,B 0,C 180,E1 -22814.079,E2 -22814.079} C_VEL
LIN {X 0,Y 227.518,Z 458.74,A -85,B 0,C 180,E1 -22814.959,E2 -22814.959} C_VEL
LIN {X 0,Y 230.603,Z 448.534,A -85,B 0,C 180,E1 -22815.585,E2 -22815.585} C_VEL
LIN {X 0,Y 233.162,Z 437.007,A -85,B 0,C 180,E1 -22816.164,E2 -22816.164} C_VEL
LIN {X 0,Y 237.434,Z 411.275,A -85,B 0,C 180,E1 -22817.213,E2 -22817.213} C_VEL
LIN {X 0,Y 236.292,Z 407.594,A -85,B 0,C 180,E1 -22819.003,E2 -22819.003} C_VEL
LIN {X 0,Y 235.503,Z 405.431,A -85,B 0,C 180,E1 -22820.378,E2 -22820.378} C_VEL
LIN {X 0,Y 234.405,Z 402.247,A -85,B 0,C 180,E1 -22823.327,E2 -22823.327} C_VEL
LIN {X 0,Y 234.029,Z 401.505,A -85,B 0,C 180,E1 -22825.211,E2 -22825.211} C_VEL
LIN {X 0,Y 234.144,Z 401.568,A -85,B 0,C 180,E1 -22828.907,E2 -22828.907} C_VEL
LIN {X 0,Y 234.636,Z 402.496,A -85,B 0,C 180,E1 -22830.74,E2 -22830.74} C_VEL
LIN {X 0,Y 235.948,Z 406.002,A -85,B 0,C 180,E1 -22833.795,E2 -22833.795} C_VEL
LIN {X 0,Y 237.212,Z 409.804,A -85,B 0,C 180,E1 -22835.919,E2 -22835.919} C_VEL
LIN {X 0,Y 232.215,Z 437.407,A -85,B 0,C 180,E1 -22837.155,E2 -22837.155} C_VEL
LIN {X 0,Y 228.465,Z 451.397,A -85,B 0,C 180,E1 -22838.098,E2 -22838.098} C_VEL
LIN {X 0,Y 225.119,Z 460.864,A -85,B 0,C 180,E1 -22838.96,E2 -22838.96} C_VEL
LIN {X 0,Y 221.261,Z 469.977,A -85,B 0,C 180,E1 -22840.035,E2 -22840.035} C_VEL
LIN {X 0,Y 216.413,Z 479.672,A -85,B 0,C 180,E1 -22841.471,E2 -22841.471} C_VEL
LIN {X 0,Y 211.486,Z 488.183,A -85,B 0,C 180,E1 -22843.097,E2 -22843.097} C_VEL
LIN {X 0,Y 205.703,Z 496.6,A -85,B 0,C 180,E1 -22845.154,E2 -22845.154} C_VEL
LIN {X 0,Y 200.247,Z 503.326,A -85,B 0,C 180,E1 -22847.34,E2 -22847.34} C_VEL
LIN {X 0,Y 195.276,Z 508.755,A -85,B 0,C 180,E1 -22849.634,E2 -22849.634} C_VEL
LIN {X 0,Y 191.543,Z 512.359,A -85,B 0,C 180,E1 -22851.562,E2 -22851.562} C_VEL
LIN {X 0,Y 186.334,Z 516.472,A -85,B 0,C 180,E1 -22854.591,E2 -22854.591} C_VEL
LIN {X 0,Y 181.853,Z 519.329,A -85,B 0,C 180,E1 -22857.786,E2 -22857.786} C_VEL
LIN {X 0,Y 179.236,Z 520.596,A -85,B 0,C 180,E1 -22860.001,E2 -22860.001} C_VEL
LIN {X 0,Y 175.985,Z 521.451,A -85,B 0,C 180,E1 -22863.279,E2 -22863.279} C_VEL
LIN {X 0,Y 173.138,Z 521.194,A -85,B 0,C 180,E1 -22866.996,E2 -22866.996} C_VEL
LIN {X 0,Y 171.367,Z 520.038,A -85,B 0,C 180,E1 -22870.179,E2 -22870.179} C_VEL
LIN {X 0,Y 170.614,Z 519.136,A -85,B 0,C 180,E1 -22871.887,E2 -22871.887} C_VEL
LIN {X 0,Y 169.499,Z 516.144,A -85,B 0,C 180,E1 -22875.637,E2 -22875.637} C_VEL
LIN {X 0,Y 169.042,Z 511.743,A -85,B 0,C 180,E1 -22879.428,E2 -22879.428} C_VEL
LIN {X 0,Y 169.153,Z 506.297,A -85,B 0,C 180,E1 -22882.981,E2 -22882.981} C_VEL
LIN {X 0,Y 169.513,Z 500.878,A -85,B 0,C 180,E1 -22885.808,E2 -22885.808} C_VEL
LIN {X 0,Y 169.994,Z 494.894,A -85,B 0,C 180,E1 -22888.39,E2 -22888.39} C_VEL
LIN {X 0,Y 170.677,Z 487.595,A -85,B 0,C 180,E1 -22891.007,E2 -22891.007} C_VEL
LIN {X 0,Y 171.591,Z 478.86,A -85,B 0,C 180,E1 -22893.57,E2 -22893.57} C_VEL
LIN {X 0,Y 172.739,Z 467.554,A -85,B 0,C 180,E1 -22896.18,E2 -22896.18} C_VEL
LIN {X 0,Y 173.796,Z 457.038,A -85,B 0,C 180,E1 -22898.076,E2 -22898.076} C_VEL
LIN {X 0,Y 174.665,Z 446.955,A -85,B 0,C 180,E1 -22899.514,E2 -22899.514} C_VEL
LIN {X 0,Y 175.532,Z 434.726,A -85,B 0,C 180,E1 -22900.838,E2 -22900.838} C_VEL
LIN {X 0,Y 176.528,Z 415.702,A -85,B 0,C 180,E1 -22902.148,E2 -22902.148} C_VEL
LIN {X 0,Y 178.428,Z 378.553,A -85,B 0,C 180,E1 -22904.445,E2 -22904.445} C_VEL
LIN {X 0,Y 175.598,Z 345.167,A -85,B 0,C 180,E1 -22906.75,E2 -22906.75} C_VEL
LIN {X 0,Y 175.502,Z 341.21,A -85,B 0,C 180,E1 -22907.014,E2 -22907.014} C_VEL
LIN {X 0,Y 175.29,Z 337.83,A -85,B 0,C 180,E1 -22908.583,E2 -22908.583} C_VEL
LIN {X 0,Y 173.243,Z 327.428,A -85,B 0,C 180,E1 -22913.694,E2 -22913.694} C_VEL
LIN {X 0,Y 171.475,Z 319.125,A -85,B 0,C 180,E1 -22918.036,E2 -22918.036} C_VEL
LIN {X 0,Y 171.367,Z 319.138,A -85,B 0,C 180,E1 -22923.182,E2 -22923.182} C_VEL
LIN {X 0,Y 171.422,Z 319.134,A -85,B 0,C 180,E1 -22928.344,E2 -22928.344} C_VEL
LIN {X 0,Y 171.515,Z 319.121,A -85,B 0,C 180,E1 -22930.861,E2 -22930.861} C_VEL
LIN {X 0,Y 171.559,Z 319.108,A -85,B 0,C 180,E1 -22935.768,E2 -22935.768} C_VEL
LIN {X 0,Y 171.849,Z 319.078,A -85,B 0,C 180,E1 -22940.581,E2 -22940.581} C_VEL
LIN {X 0,Y 171.783,Z 319.082,A -85,B 0,C 180,E1 -22945.302,E2 -22945.302} C_VEL
LIN {X 0,Y 172.313,Z 319.021,A -85,B 0,C 180,E1 -22949.995,E2 -22949.995} C_VEL
LIN {X 0,Y 171.86,Z 319.075,A -85,B 0,C 180,E1 -22957.041,E2 -22957.041} C_VEL
LIN {X 0,Y 171.769,Z 319.085,A -85,B 0,C 180,E1 -22960.889,E2 -22960.889} C_VEL
LIN {X 0,Y 171.519,Z 319.121,A -85,B 0,C 180,E1 -22966.661,E2 -22966.661} C_VEL
LIN {X 0,Y 171.42,Z 319.125,A -85,B 0,C 180,E1 -22971.646,E2 -22971.646} C_VEL
LIN {X 0,Y 171.438,Z 319.13,A -85,B 0,C 180,E1 -22975.591,E2 -22975.591} C_VEL
LIN {X 0,Y 171.408,Z 319.126,A -85,B 0,C 180,E1 -22980.565,E2 -22980.565} C_VEL
LIN {X 0,Y 171.381,Z 319.136,A -85,B 0,C 180,E1 -22985.028,E2 -22985.028} C_VEL
LIN {X 0,Y 171.33,Z 319.137,A -85,B 0,C 180,E1 -22988.794,E2 -22988.794} C_VEL
LIN {X 0,Y 171.303,Z 319.148,A -85,B 0,C 180,E1 -22994.211,E2 -22994.211} C_VEL
LIN {X 0,Y 171.311,Z 319.142,A -85,B 0,C 180,E1 -22998.973,E2 -22998.973} C_VEL
LIN {X 0,Y 171.339,Z 319.141,A -85,B 0,C 180,E1 -23002.027,E2 -23002.027} C_VEL
LIN {X 0,Y 171.376,Z 319.135,A -85,B 0,C 180,E1 -23005.087,E2 -23005.087} C_VEL
LIN {X 0,Y 171.424,Z 319.13,A -85,B 0,C 180,E1 -23010.528,E2 -23010.528} C_VEL
LIN {X 0,Y 171.411,Z 319.128,A -85,B 0,C 180,E1 -23015.793,E2 -23015.793} C_VEL
LIN {X 0,Y 171.478,Z 319.123,A -85,B 0,C 180,E1 -23020.859,E2 -23020.859} C_VEL
LIN {X 0,Y 171.519,Z 319.114,A -85,B 0,C 180,E1 -23025.767,E2 -23025.767} C_VEL
LIN {X 0,Y 171.811,Z 319.083,A -85,B 0,C 180,E1 -23030.582,E2 -23030.582} C_VEL
LIN {X 0,Y 171.777,Z 319.084,A -85,B 0,C 180,E1 -23035.305,E2 -23035.305} C_VEL
LIN {X 0,Y 172.293,Z 319.021,A -85,B 0,C 180,E1 -23039.999,E2 -23039.999} C_VEL
LIN {X 0,Y 171.772,Z 319.085,A -85,B 0,C 180,E1 -23044.692,E2 -23044.692} C_VEL
LIN {X 0,Y 171.812,Z 319.082,A -85,B 0,C 180,E1 -23049.416,E2 -23049.416} C_VEL
LIN {X 0,Y 171.534,Z 319.116,A -85,B 0,C 180,E1 -23054.229,E2 -23054.229} C_VEL
LIN {X 0,Y 171.508,Z 319.118,A -85,B 0,C 180,E1 -23059.557,E2 -23059.557} C_VEL
LIN {X 0,Y 171.419,Z 319.131,A -85,B 0,C 180,E1 -23065.604,E2 -23065.604} C_VEL
LIN {X 0,Y 171.392,Z 319.131,A -85,B 0,C 180,E1 -23070.577,E2 -23070.577} C_VEL
LIN {X 0,Y 171.366,Z 319.139,A -85,B 0,C 180,E1 -23075.04,E2 -23075.04} C_VEL
LIN {X 0,Y 171.318,Z 319.147,A -85,B 0,C 180,E1 -23078.806,E2 -23078.806} C_VEL
LIN {X 0,Y 171.297,Z 319.147,A -85,B 0,C 180,E1 -23084.223,E2 -23084.223} C_VEL
LIN {X 0,Y 171.411,Z 319.293,A -85,B 0,C 180,E1 -23088.343,E2 -23088.343} C_VEL
LIN {X 0,Y 173.618,Z 329.051,A -85,B 0,C 180,E1 -23093.041,E2 -23093.041} C_VEL
LIN {X 0,Y 175.95,Z 340.014,A -85,B 0,C 180,E1 -23098.02,E2 -23098.02} C_VEL
LIN {X 0,Y 176.709,Z 343.698,A -85,B 0,C 180,E1 -23099.608,E2 -23099.608} C_VEL
LIN {X 0,Y 177.7,Z 348.615,A -85,B 0,C 180,E1 -23099.968,E2 -23099.968} C_VEL
LIN {X 0,Y 179.044,Z 374.1,A -85,B 0,C 180,E1 -23101.55,E2 -23101.55} C_VEL
LIN {X 0,Y 179.723,Z 384.29,A -85,B 0,C 180,E1 -23102.181,E2 -23102.181} C_VEL
LIN {X 0,Y 177.13,Z 442.064,A -85,B 0,C 180,E1 -23105.474,E2 -23105.474} C_VEL
LIN {X 0,Y 176.484,Z 452,A -85,B 0,C 180,E1 -23106.289,E2 -23106.289} C_VEL
LIN {X 0,Y 175.575,Z 462.112,A -85,B 0,C 180,E1 -23107.412,E2 -23107.412} C_VEL
LIN {X 0,Y 174.604,Z 471.582,A -85,B 0,C 180,E1 -23108.768,E2 -23108.768} C_VEL
LIN {X 0,Y 173.735,Z 479.75,A -85,B 0,C 180,E1 -23110.204,E2 -23110.204} C_VEL
LIN {X 0,Y 172.812,Z 487.975,A -85,B 0,C 180,E1 -23111.942,E2 -23111.942} C_VEL
LIN {X 0,Y 171.933,Z 495.533,A -85,B 0,C 180,E1 -23113.842,E2 -23113.842} C_VEL
LIN {X 0,Y 170.872,Z 499.982,A -85,B 0,C 180,E1 -23115.139,E2 -23115.139} C_VEL
LIN {X 0,Y 168.893,Z 503.931,A -85,B 0,C 180,E1 -23116.474,E2 -23116.474} C_VEL
LIN {X 0,Y 163.988,Z 512.22,A -85,B 0,C 180,E1 -23119.93,E2 -23119.93} C_VEL
LIN {X 0,Y 163.141,Z 515.588,A -85,B 0,C 180,E1 -23121.621,E2 -23121.621} C_VEL
LIN {X 0,Y 163.036,Z 521.826,A -85,B 0,C 180,E1 -23125.06,E2 -23125.06} C_VEL
LIN {X 0,Y 163.004,Z 525.536,A -85,B 0,C 180,E1 -23127.534,E2 -23127.534} C_VEL
LIN {X 0,Y 163.095,Z 528.503,A -85,B 0,C 180,E1 -23130.005,E2 -23130.005} C_VEL
LIN {X 0,Y 162.724,Z 530.886,A -85,B 0,C 180,E1 -23132.48,E2 -23132.48} C_VEL
LIN {X 0,Y 162.412,Z 533.194,A -85,B 0,C 180,E1 -23135.587,E2 -23135.587} C_VEL
LIN {X 0,Y 162.544,Z 535.235,A -85,B 0,C 180,E1 -23139.963,E2 -23139.963} C_VEL
LIN {X 0,Y 163.042,Z 535.931,A -85,B 0,C 180,E1 -23142.45,E2 -23142.45} C_VEL
LIN {X 0,Y 165.023,Z 536.072,A -85,B 0,C 180,E1 -23147.348,E2 -23147.348} C_VEL
LIN {X 0,Y 168.48,Z 534.664,A -85,B 0,C 180,E1 -23152.054,E2 -23152.054} C_VEL
LIN {X 0,Y 170.696,Z 533.492,A -85,B 0,C 180,E1 -23154.316,E2 -23154.316} C_VEL
LIN {X 0,Y 175.847,Z 529.736,A -85,B 0,C 180,E1 -23158.661,E2 -23158.661} C_VEL
LIN {X 0,Y 180.665,Z 525.844,A -85,B 0,C 180,E1 -23161.681,E2 -23161.681} C_VEL
LIN {X 0,Y 186.116,Z 520.836,A -85,B 0,C 180,E1 -23164.502,E2 -23164.502} C_VEL
LIN {X 0,Y 191.008,Z 515.808,A -85,B 0,C 180,E1 -23166.721,E2 -23166.721} C_VEL
LIN {X 0,Y 196.357,Z 509.784,A -85,B 0,C 180,E1 -23168.783,E2 -23168.783} C_VEL
LIN {X 0,Y 201.988,Z 502.571,A -85,B 0,C 180,E1 -23170.722,E2 -23170.722} C_VEL
LIN {X 0,Y 206.696,Z 495.804,A -85,B 0,C 180,E1 -23172.185,E2 -23172.185} C_VEL
LIN {X 0,Y 212.257,Z 486.806,A -85,B 0,C 180,E1 -23173.724,E2 -23173.724} C_VEL
LIN {X 0,Y 216.733,Z 478.507,A -85,B 0,C 180,E1 -23174.852,E2 -23174.852} C_VEL
LIN {X 0,Y 221.424,Z 468.363,A -85,B 0,C 180,E1 -23175.899,E2 -23175.899} C_VEL
LIN {X 0,Y 224.993,Z 459.134,A -85,B 0,C 180,E1 -23176.638,E2 -23176.638} C_VEL
LIN {X 0,Y 228.024,Z 449.633,A -85,B 0,C 180,E1 -23177.217,E2 -23177.217} C_VEL
LIN {X 0,Y 230.818,Z 438.065,A -85,B 0,C 180,E1 -23177.799,E2 -23177.799} C_VEL
LIN {X 0,Y 234.867,Z 415.608,A -85,B 0,C 180,E1 -23178.695,E2 -23178.695} C_VEL
LIN {X 0,Y 233.797,Z 412.199,A -85,B 0,C 180,E1 -23180.693,E2 -23180.693} C_VEL
LIN {X 0,Y 232.765,Z 408.953,A -85,B 0,C 180,E1 -23183.814,E2 -23183.814} C_VEL
LIN {X 0,Y 232.574,Z 408.493,A -85,B 0,C 180,E1 -23184.961,E2 -23184.961} C_VEL
LIN {X 0,Y 232.58,Z 408.42,A -85,B 0,C 180,E1 -23188.554,E2 -23188.554} C_VEL
LIN {X 0,Y 232.954,Z 409.11,A -85,B 0,C 180,E1 -23190.273,E2 -23190.273} C_VEL
LIN {X 0,Y 234.097,Z 412.704,A -85,B 0,C 180,E1 -23193.393,E2 -23193.393} C_VEL
LIN {X 0,Y 234.658,Z 414.415,A -85,B 0,C 180,E1 -23194.43,E2 -23194.43} C_VEL
LIN {X 0,Y 230.037,Z 438.39,A -85,B 0,C 180,E1 -23195.503,E2 -23195.503} C_VEL
LIN {X 0,Y 226.153,Z 451.916,A -85,B 0,C 180,E1 -23196.401,E2 -23196.401} C_VEL
LIN {X 0,Y 222.077,Z 462.803,A -85,B 0,C 180,E1 -23197.392,E2 -23197.392} C_VEL
LIN {X 0,Y 217.939,Z 471.975,A -85,B 0,C 180,E1 -23198.481,E2 -23198.481} C_VEL
LIN {X 0,Y 212.695,Z 481.73,A -85,B 0,C 180,E1 -23199.952,E2 -23199.952} C_VEL
LIN {X 0,Y 206.628,Z 491.102,A -85,B 0,C 180,E1 -23201.846,E2 -23201.846} C_VEL
LIN {X 0,Y 200.989,Z 498.521,A -85,B 0,C 180,E1 -23203.757,E2 -23203.757} C_VEL
LIN {X 0,Y 195.761,Z 504.523,A -85,B 0,C 180,E1 -23205.766,E2 -23205.766} C_VEL
LIN {X 0,Y 190.05,Z 510.158,A -85,B 0,C 180,E1 -23208.266,E2 -23208.266} C_VEL
LIN {X 0,Y 185.148,Z 514.319,A -85,B 0,C 180,E1 -23210.719,E2 -23210.719} C_VEL
LIN {X 0,Y 180.636,Z 517.516,A -85,B 0,C 180,E1 -23213.298,E2 -23213.298} C_VEL
LIN {X 0,Y 176.04,Z 520.073,A -85,B 0,C 180,E1 -23216.419,E2 -23216.419} C_VEL
LIN {X 0,Y 174.42,Z 520.858,A -85,B 0,C 180,E1 -23217.692,E2 -23217.692} C_VEL
LIN {X 0,Y 171.765,Z 521.661,A -85,B 0,C 180,E1 -23220.001,E2 -23220.001} C_VEL
LIN {X 0,Y 168.899,Z 522.004,A -85,B 0,C 180,E1 -23222.991,E2 -23222.991} C_VEL
LIN {X 0,Y 165.702,Z 521.26,A -85,B 0,C 180,E1 -23227.311,E2 -23227.311} C_VEL
LIN {X 0,Y 164.2,Z 519.892,A -85,B 0,C 180,E1 -23230.127,E2 -23230.127} C_VEL
LIN {X 0,Y 162.848,Z 517.322,A -85,B 0,C 180,E1 -23233.732,E2 -23233.732} C_VEL
LIN {X 0,Y 162.098,Z 513.351,A -85,B 0,C 180,E1 -23237.669,E2 -23237.669} C_VEL
LIN {X 0,Y 162.004,Z 507.844,A -85,B 0,C 180,E1 -23241.64,E2 -23241.64} C_VEL
LIN {X 0,Y 162.345,Z 501.944,A -85,B 0,C 180,E1 -23244.95,E2 -23244.95} C_VEL
LIN {X 0,Y 162.793,Z 496.074,A -85,B 0,C 180,E1 -23247.653,E2 -23247.653} C_VEL
LIN {X 0,Y 163.394,Z 489.455,A -85,B 0,C 180,E1 -23250.2,E2 -23250.2} C_VEL
LIN {X 0,Y 164.181,Z 481.606,A -85,B 0,C 180,E1 -23252.715,E2 -23252.715} C_VEL
LIN {X 0,Y 165.131,Z 472.689,A -85,B 0,C 180,E1 -23255.071,E2 -23255.071} C_VEL
LIN {X 0,Y 166.261,Z 461.674,A -85,B 0,C 180,E1 -23257.421,E2 -23257.421} C_VEL
LIN {X 0,Y 167.282,Z 450.27,A -85,B 0,C 180,E1 -23259.26,E2 -23259.26} C_VEL
LIN {X 0,Y 168.216,Z 439.677,A -85,B 0,C 180,E1 -23260.558,E2 -23260.558} C_VEL
LIN {X 0,Y 168.839,Z 429.315,A -85,B 0,C 180,E1 -23261.502,E2 -23261.502} C_VEL
LIN {X 0,Y 171.375,Z 378.453,A -85,B 0,C 180,E1 -23264.843,E2 -23264.843} C_VEL
LIN {X 0,Y 168.615,Z 344.876,A -85,B 0,C 180,E1 -23267.263,E2 -23267.263} C_VEL
LIN {X 0,Y 168.509,Z 341.229,A -85,B 0,C 180,E1 -23267.534,E2 -23267.534} C_VEL
LIN {X 0,Y 167.564,Z 335.422,A -85,B 0,C 180,E1 -23270.41,E2 -23270.41} C_VEL
LIN {X 0,Y 165.784,Z 326.364,A -85,B 0,C 180,E1 -23275.087,E2 -23275.087} C_VEL
LIN {X 0,Y 164.415,Z 320.004,A -85,B 0,C 180,E1 -23278.593,E2 -23278.593} C_VEL
LIN {X 0,Y 164.362,Z 320.012,A -85,B 0,C 180,E1 -23284.682,E2 -23284.682} C_VEL
LIN {X 0,Y 164.423,Z 320.003,A -85,B 0,C 180,E1 -23290.115,E2 -23290.115} C_VEL
LIN {X 0,Y 164.487,Z 319.99,A -85,B 0,C 180,E1 -23295.142,E2 -23295.142} C_VEL
LIN {X 0,Y 164.77,Z 319.959,A -85,B 0,C 180,E1 -23300.173,E2 -23300.173} C_VEL
LIN {X 0,Y 164.824,Z 319.952,A -85,B 0,C 180,E1 -23302.646,E2 -23302.646} C_VEL
LIN {X 0,Y 165.277,Z 319.897,A -85,B 0,C 180,E1 -23309.995,E2 -23309.995} C_VEL
LIN {X 0,Y 164.822,Z 319.952,A -85,B 0,C 180,E1 -23317.344,E2 -23317.344} C_VEL
LIN {X 0,Y 164.703,Z 319.965,A -85,B 0,C 180,E1 -23321.053,E2 -23321.053} C_VEL
LIN {X 0,Y 164.437,Z 320.001,A -85,B 0,C 180,E1 -23327.401,E2 -23327.401} C_VEL
LIN {X 0,Y 164.347,Z 320.007,A -85,B 0,C 180,E1 -23332.628,E2 -23332.628} C_VEL
LIN {X 0,Y 164.364,Z 320.01,A -85,B 0,C 180,E1 -23336.109,E2 -23336.109} C_VEL
LIN {X 0,Y 164.348,Z 320.007,A -85,B 0,C 180,E1 -23341.209,E2 -23341.209} C_VEL
LIN {X 0,Y 164.268,Z 320.02,A -85,B 0,C 180,E1 -23346.786,E2 -23346.786} C_VEL
LIN {X 0,Y 164.272,Z 320.017,A -85,B 0,C 180,E1 -23349.91,E2 -23349.91} C_VEL
LIN {X 0,Y 164.265,Z 320.022,A -85,B 0,C 180,E1 -23353.334,E2 -23353.334} C_VEL
LIN {X 0,Y 164.243,Z 320.022,A -85,B 0,C 180,E1 -23356.791,E2 -23356.791} C_VEL
LIN {X 0,Y 164.27,Z 320.02,A -85,B 0,C 180,E1 -23360.348,E2 -23360.348} C_VEL
LIN {X 0,Y 164.304,Z 320.014,A -85,B 0,C 180,E1 -23366.214,E2 -23366.214} C_VEL
LIN {X 0,Y 164.366,Z 320.008,A -85,B 0,C 180,E1 -23369.128,E2 -23369.128} C_VEL
LIN {X 0,Y 164.379,Z 320.005,A -85,B 0,C 180,E1 -23374.686,E2 -23374.686} C_VEL
LIN {X 0,Y 164.389,Z 320.008,A -85,B 0,C 180,E1 -23380.113,E2 -23380.113} C_VEL
LIN {X 0,Y 164.448,Z 319.993,A -85,B 0,C 180,E1 -23385.141,E2 -23385.141} C_VEL
LIN {X 0,Y 164.733,Z 319.966,A -85,B 0,C 180,E1 -23390.173,E2 -23390.173} C_VEL
LIN {X 0,Y 164.793,Z 319.953,A -85,B 0,C 180,E1 -23392.648,E2 -23392.648} C_VEL
LIN {X 0,Y 165.012,Z 319.929,A -85,B 0,C 180,E1 -23397.558,E2 -23397.558} C_VEL
LIN {X 0,Y 165.256,Z 319.898,A -85,B 0,C 180,E1 -23399.999,E2 -23399.999} C_VEL
LIN {X 0,Y 164.721,Z 319.964,A -85,B 0,C 180,E1 -23404.894,E2 -23404.894} C_VEL
LIN {X 0,Y 164.793,Z 319.959,A -85,B 0,C 180,E1 -23407.349,E2 -23407.349} C_VEL
LIN {X 0,Y 164.671,Z 319.969,A -85,B 0,C 180,E1 -23411.058,E2 -23411.058} C_VEL
LIN {X 0,Y 164.446,Z 320,A -85,B 0,C 180,E1 -23417.406,E2 -23417.406} C_VEL
LIN {X 0,Y 164.444,Z 319.997,A -85,B 0,C 180,E1 -23419.992,E2 -23419.992} C_VEL
LIN {X 0,Y 164.346,Z 320.014,A -85,B 0,C 180,E1 -23426.122,E2 -23426.122} C_VEL
LIN {X 0,Y 164.331,Z 320.013,A -85,B 0,C 180,E1 -23431.221,E2 -23431.221} C_VEL
LIN {X 0,Y 164.254,Z 320.024,A -85,B 0,C 180,E1 -23436.798,E2 -23436.798} C_VEL
LIN {X 0,Y 164.262,Z 320.024,A -85,B 0,C 180,E1 -23439.923,E2 -23439.923} C_VEL
LIN {X 0,Y 164.258,Z 320.026,A -85,B 0,C 180,E1 -23443.347,E2 -23443.347} C_VEL
LIN {X 0,Y 164.316,Z 320.201,A -85,B 0,C 180,E1 -23447.768,E2 -23447.768} C_VEL
LIN {X 0,Y 166.429,Z 329.395,A -85,B 0,C 180,E1 -23452.393,E2 -23452.393} C_VEL
LIN {X 0,Y 168.965,Z 341.255,A -85,B 0,C 180,E1 -23458.014,E2 -23458.014} C_VEL
LIN {X 0,Y 169.453,Z 343.537,A -85,B 0,C 180,E1 -23459.061,E2 -23459.061} C_VEL
LIN {X 0,Y 170.767,Z 349.865,A -85,B 0,C 180,E1 -23459.564,E2 -23459.564} C_VEL
LIN {X 0,Y 172.225,Z 376.87,A -85,B 0,C 180,E1 -23461.32,E2 -23461.32} C_VEL
LIN {X 0,Y 172.675,Z 385.219,A -85,B 0,C 180,E1 -23461.852,E2 -23461.852} C_VEL
LIN {X 0,Y 170.063,Z 442.341,A -85,B 0,C 180,E1 -23465.269,E2 -23465.269} C_VEL
LIN {X 0,Y 169.368,Z 452.364,A -85,B 0,C 180,E1 -23466.143,E2 -23466.143} C_VEL
LIN {X 0,Y 168.452,Z 462.186,A -85,B 0,C 180,E1 -23467.297,E2 -23467.297} C_VEL
LIN {X 0,Y 167.452,Z 471.97,A -85,B 0,C 180,E1 -23468.785,E2 -23468.785} C_VEL
LIN {X 0,Y 166.445,Z 481.421,A -85,B 0,C 180,E1 -23470.586,E2 -23470.586} C_VEL
LIN {X 0,Y 165.346,Z 490.426,A -85,B 0,C 180,E1 -23472.697,E2 -23472.697} C_VEL
LIN {X 0,Y 164.431,Z 499.012,A -85,B 0,C 180,E1 -23475.147,E2 -23475.147} C_VEL
LIN {X 0,Y 163.573,Z 507.844,A -85,B 0,C 180,E1 -23478.23,E2 -23478.23} C_VEL
LIN {X 0,Y 163.141,Z 515.588,A -85,B 0,C 180,E1 -23481.621,E2 -23481.621} C_VEL
LIN {X 0,Y 162.446,Z 518.794,A -85,B 0,C 180,E1 -23483.372,E2 -23483.372} C_VEL
LIN {X 0,Y 160.94,Z 521.562,A -85,B 0,C 180,E1 -23485.163,E2 -23485.163} C_VEL
LIN {X 0,Y 157.321,Z 526.1,A -85,B 0,C 180,E1 -23488.946,E2 -23488.946} C_VEL
LIN {X 0,Y 155.904,Z 528.73,A -85,B 0,C 180,E1 -23491.661,E2 -23491.661} C_VEL
LIN {X 0,Y 155.419,Z 532.08,A -85,B 0,C 180,E1 -23495.839,E2 -23495.839} C_VEL
LIN {X 0,Y 155.564,Z 534.427,A -85,B 0,C 180,E1 -23500.415,E2 -23500.415} C_VEL
LIN {X 0,Y 157.024,Z 535.558,A -85,B 0,C 180,E1 -23505.582,E2 -23505.582} C_VEL
LIN {X 0,Y 158.254,Z 535.634,A -85,B 0,C 180,E1 -23508.115,E2 -23508.115} C_VEL
LIN {X 0,Y 161.908,Z 534.608,A -85,B 0,C 180,E1 -23512.999,E2 -23512.999} C_VEL
LIN {X 0,Y 166.781,Z 532.012,A -85,B 0,C 180,E1 -23517.618,E2 -23517.618} C_VEL
LIN {X 0,Y 171.321,Z 529.064,A -85,B 0,C 180,E1 -23520.851,E2 -23520.851} C_VEL
LIN {X 0,Y 176.504,Z 525.145,A -85,B 0,C 180,E1 -23523.881,E2 -23523.881} C_VEL
LIN {X 0,Y 182.356,Z 520.168,A -85,B 0,C 180,E1 -23526.683,E2 -23526.683} C_VEL
LIN {X 0,Y 187.636,Z 515.1,A -85,B 0,C 180,E1 -23528.858,E2 -23528.858} C_VEL
LIN {X 0,Y 194.433,Z 507.657,A -85,B 0,C 180,E1 -23531.275,E2 -23531.275} C_VEL
LIN {X 0,Y 200.48,Z 500.212,A -85,B 0,C 180,E1 -23533.125,E2 -23533.125} C_VEL
LIN {X 0,Y 205.506,Z 493.172,A -85,B 0,C 180,E1 -23534.513,E2 -23534.513} C_VEL
LIN {X 0,Y 210.646,Z 484.92,A -85,B 0,C 180,E1 -23535.834,E2 -23535.834} C_VEL
LIN {X 0,Y 215.364,Z 476.289,A -85,B 0,C 180,E1 -23536.9,E2 -23536.9} C_VEL
LIN {X 0,Y 220.005,Z 466.481,A -85,B 0,C 180,E1 -23537.843,E2 -23537.843} C_VEL
LIN {X 0,Y 224.58,Z 454.704,A -85,B 0,C 180,E1 -23538.681,E2 -23538.681} C_VEL
LIN {X 0,Y 228.509,Z 440.883,A -85,B 0,C 180,E1 -23539.387,E2 -23539.387} C_VEL
LIN {X 0,Y 232.441,Z 420.335,A -85,B 0,C 180,E1 -23540.218,E2 -23540.218} C_VEL
LIN {X 0,Y 231.958,Z 418.479,A -85,B 0,C 180,E1 -23541.448,E2 -23541.448} C_VEL
LIN {X 0,Y 231.242,Z 415.847,A -85,B 0,C 180,E1 -23543.966,E2 -23543.966} C_VEL
LIN {X 0,Y 231.036,Z 415.4,A -85,B 0,C 180,E1 -23545.216,E2 -23545.216} C_VEL
LIN {X 0,Y 231.126,Z 415.438,A -85,B 0,C 180,E1 -23548.875,E2 -23548.875} C_VEL
LIN {X 0,Y 231.338,Z 416.015,A -85,B 0,C 180,E1 -23550.044,E2 -23550.044} C_VEL
LIN {X 0,Y 232.231,Z 419.262,A -85,B 0,C 180,E1 -23552.899,E2 -23552.899} C_VEL
LIN {X 0,Y 228.053,Z 439.985,A -85,B 0,C 180,E1 -23553.837,E2 -23553.837} C_VEL
LIN {X 0,Y 224.072,Z 453.006,A -85,B 0,C 180,E1 -23554.702,E2 -23554.702} C_VEL
LIN {X 0,Y 220.416,Z 462.346,A -85,B 0,C 180,E1 -23555.513,E2 -23555.513} C_VEL
LIN {X 0,Y 216.271,Z 471.195,A -85,B 0,C 180,E1 -23556.515,E2 -23556.515} C_VEL
LIN {X 0,Y 211.507,Z 479.762,A -85,B 0,C 180,E1 -23557.716,E2 -23557.716} C_VEL
LIN {X 0,Y 206.658,Z 487.442,A -85,B 0,C 180,E1 -23559.08,E2 -23559.08} C_VEL
LIN {X 0,Y 200.878,Z 495.303,A -85,B 0,C 180,E1 -23560.841,E2 -23560.841} C_VEL
LIN {X 0,Y 194.044,Z 503.188,A -85,B 0,C 180,E1 -23563.158,E2 -23563.158} C_VEL
LIN {X 0,Y 187.142,Z 509.796,A -85,B 0,C 180,E1 -23565.871,E2 -23565.871} C_VEL
LIN {X 0,Y 180.79,Z 514.852,A -85,B 0,C 180,E1 -23568.793,E2 -23568.793} C_VEL
LIN {X 0,Y 176.869,Z 517.466,A -85,B 0,C 180,E1 -23570.856,E2 -23570.856} C_VEL
LIN {X 0,Y 173.272,Z 519.576,A -85,B 0,C 180,E1 -23573.012,E2 -23573.012} C_VEL
LIN {X 0,Y 169.103,Z 521.403,A -85,B 0,C 180,E1 -23575.894,E2 -23575.894} C_VEL
LIN {X 0,Y 164.27,Z 522.471,A -85,B 0,C 180,E1 -23580.001,E2 -23580.001} C_VEL
LIN {X 0,Y 161.814,Z 522.496,A -85,B 0,C 180,E1 -23582.645,E2 -23582.645} C_VEL
LIN {X 0,Y 159.927,Z 521.938,A -85,B 0,C 180,E1 -23585.044,E2 -23585.044} C_VEL
LIN {X 0,Y 157.044,Z 519.581,A -85,B 0,C 180,E1 -23590.09,E2 -23590.09} C_VEL
LIN {X 0,Y 155.927,Z 517.407,A -85,B 0,C 180,E1 -23593.026,E2 -23593.026} C_VEL
LIN {X 0,Y 155.015,Z 512.342,A -85,B 0,C 180,E1 -23597.809,E2 -23597.809} C_VEL
LIN {X 0,Y 154.93,Z 507.525,A -85,B 0,C 180,E1 -23601.28,E2 -23601.28} C_VEL
LIN {X 0,Y 155.156,Z 502.84,A -85,B 0,C 180,E1 -23604.06,E2 -23604.06} C_VEL
LIN {X 0,Y 155.597,Z 497.225,A -85,B 0,C 180,E1 -23606.853,E2 -23606.853} C_VEL
LIN {X 0,Y 156.169,Z 490.328,A -85,B 0,C 180,E1 -23609.673,E2 -23609.673} C_VEL
LIN {X 0,Y 156.898,Z 482.952,A -85,B 0,C 180,E1 -23612.187,E2 -23612.187} C_VEL
LIN {X 0,Y 157.845,Z 474.454,A -85,B 0,C 180,E1 -23614.591,E2 -23614.591} C_VEL
LIN {X 0,Y 158.787,Z 465.051,A -85,B 0,C 180,E1 -23616.772,E2 -23616.772} C_VEL
LIN {X 0,Y 159.94,Z 453.121,A -85,B 0,C 180,E1 -23618.972,E2 -23618.972} C_VEL
LIN {X 0,Y 160.97,Z 441.831,A -85,B 0,C 180,E1 -23620.502,E2 -23620.502} C_VEL
LIN {X 0,Y 161.64,Z 430.758,A -85,B 0,C 180,E1 -23621.612,E2 -23621.612} C_VEL
LIN {X 0,Y 164.45,Z 379.841,A -85,B 0,C 180,E1 -23625.157,E2 -23625.157} C_VEL
LIN {X 0,Y 161.675,Z 345.565,A -85,B 0,C 180,E1 -23627.723,E2 -23627.723} C_VEL
LIN {X 0,Y 161.485,Z 341.298,A -85,B 0,C 180,E1 -23628.054,E2 -23628.054} C_VEL
LIN {X 0,Y 159.771,Z 332.459,A -85,B 0,C 180,E1 -23632.671,E2 -23632.671} C_VEL
LIN {X 0,Y 157.872,Z 323.256,A -85,B 0,C 180,E1 -23637.763,E2 -23637.763} C_VEL
LIN {X 0,Y 157.349,Z 320.884,A -85,B 0,C 180,E1 -23639.118,E2 -23639.118} C_VEL
LIN {X 0,Y 157.273,Z 320.894,A -85,B 0,C 180,E1 -23643.454,E2 -23643.454} C_VEL
LIN {X 0,Y 157.366,Z 320.882,A -85,B 0,C 180,E1 -23649.7,E2 -23649.7} C_VEL
LIN {X 0,Y 157.42,Z 320.874,A -85,B 0,C 180,E1 -23654.459,E2 -23654.459} C_VEL
LIN {X 0,Y 157.693,Z 320.841,A -85,B 0,C 180,E1 -23659.727,E2 -23659.727} C_VEL
LIN {X 0,Y 157.763,Z 320.831,A -85,B 0,C 180,E1 -23662.315,E2 -23662.315} C_VEL
LIN {X 0,Y 158.239,Z 320.774,A -85,B 0,C 180,E1 -23669.995,E2 -23669.995} C_VEL
LIN {X 0,Y 157.76,Z 320.832,A -85,B 0,C 180,E1 -23677.674,E2 -23677.674} C_VEL
LIN {X 0,Y 157.633,Z 320.845,A -85,B 0,C 180,E1 -23681.222,E2 -23681.222} C_VEL
LIN {X 0,Y 157.417,Z 320.874,A -85,B 0,C 180,E1 -23685.531,E2 -23685.531} C_VEL
LIN {X 0,Y 157.307,Z 320.885,A -85,B 0,C 180,E1 -23690.934,E2 -23690.934} C_VEL
LIN {X 0,Y 157.304,Z 320.89,A -85,B 0,C 180,E1 -23696.673,E2 -23696.673} C_VEL
LIN {X 0,Y 157.258,Z 320.893,A -85,B 0,C 180,E1 -23702.422,E2 -23702.422} C_VEL
LIN {X 0,Y 157.247,Z 320.896,A -85,B 0,C 180,E1 -23706.436,E2 -23706.436} C_VEL
LIN {X 0,Y 157.175,Z 320.905,A -85,B 0,C 180,E1 -23712.11,E2 -23712.11} C_VEL
LIN {X 0,Y 157.172,Z 320.902,A -85,B 0,C 180,E1 -23717.875,E2 -23717.875} C_VEL
LIN {X 0,Y 157.238,Z 320.897,A -85,B 0,C 180,E1 -23723.549,E2 -23723.549} C_VEL
LIN {X 0,Y 157.27,Z 320.889,A -85,B 0,C 180,E1 -23728.091,E2 -23728.091} C_VEL
LIN {X 0,Y 157.289,Z 320.891,A -85,B 0,C 180,E1 -23733.459,E2 -23733.459} C_VEL
LIN {X 0,Y 157.333,Z 320.887,A -85,B 0,C 180,E1 -23739.698,E2 -23739.698} C_VEL
LIN {X 0,Y 157.381,Z 320.874,A -85,B 0,C 180,E1 -23744.457,E2 -23744.457} C_VEL
LIN {X 0,Y 157.656,Z 320.846,A -85,B 0,C 180,E1 -23749.727,E2 -23749.727} C_VEL
LIN {X 0,Y 157.73,Z 320.835,A -85,B 0,C 180,E1 -23752.317,E2 -23752.317} C_VEL
LIN {X 0,Y 158.219,Z 320.774,A -85,B 0,C 180,E1 -23759.999,E2 -23759.999} C_VEL
LIN {X 0,Y 157.73,Z 320.837,A -85,B 0,C 180,E1 -23767.68,E2 -23767.68} C_VEL
LIN {X 0,Y 157.602,Z 320.849,A -85,B 0,C 180,E1 -23771.226,E2 -23771.226} C_VEL
LIN {X 0,Y 157.404,Z 320.878,A -85,B 0,C 180,E1 -23775.538,E2 -23775.538} C_VEL
LIN {X 0,Y 157.337,Z 320.88,A -85,B 0,C 180,E1 -23780.936,E2 -23780.936} C_VEL
LIN {X 0,Y 157.283,Z 320.892,A -85,B 0,C 180,E1 -23786.684,E2 -23786.684} C_VEL
LIN {X 0,Y 157.242,Z 320.897,A -85,B 0,C 180,E1 -23792.434,E2 -23792.434} C_VEL
LIN {X 0,Y 157.233,Z 320.897,A -85,B 0,C 180,E1 -23796.448,E2 -23796.448} C_VEL
LIN {X 0,Y 157.167,Z 320.907,A -85,B 0,C 180,E1 -23802.123,E2 -23802.123} C_VEL
LIN {X 0,Y 157.256,Z 320.975,A -85,B 0,C 180,E1 -23807.105,E2 -23807.105} C_VEL
LIN {X 0,Y 159.56,Z 331.161,A -85,B 0,C 180,E1 -23812.449,E2 -23812.449} C_VEL
LIN {X 0,Y 161.903,Z 342.214,A -85,B 0,C 180,E1 -23817.887,E2 -23817.887} C_VEL
LIN {X 0,Y 162.243,Z 343.79,A -85,B 0,C 180,E1 -23818.554,E2 -23818.554} C_VEL
LIN {X 0,Y 163.818,Z 350.332,A -85,B 0,C 180,E1 -23819.093,E2 -23819.093} C_VEL
LIN {X 0,Y 165.108,Z 375.292,A -85,B 0,C 180,E1 -23820.782,E2 -23820.782} C_VEL
LIN {X 0,Y 165.733,Z 384.3,A -85,B 0,C 180,E1 -23821.393,E2 -23821.393} C_VEL
LIN {X 0,Y 163.022,Z 441.951,A -85,B 0,C 180,E1 -23825.046,E2 -23825.046} C_VEL
LIN {X 0,Y 162.281,Z 452.279,A -85,B 0,C 180,E1 -23825.997,E2 -23825.997} C_VEL
LIN {X 0,Y 161.315,Z 462.4,A -85,B 0,C 180,E1 -23827.261,E2 -23827.261} C_VEL
LIN {X 0,Y 160.341,Z 472.02,A -85,B 0,C 180,E1 -23828.808,E2 -23828.808} C_VEL
LIN {X 0,Y 159.31,Z 481.377,A -85,B 0,C 180,E1 -23830.686,E2 -23830.686} C_VEL
LIN {X 0,Y 158.218,Z 490.327,A -85,B 0,C 180,E1 -23832.893,E2 -23832.893} C_VEL
LIN {X 0,Y 157.432,Z 497.863,A -85,B 0,C 180,E1 -23835.133,E2 -23835.133} C_VEL
LIN {X 0,Y 156.725,Z 505.133,A -85,B 0,C 180,E1 -23837.708,E2 -23837.708} C_VEL
LIN {X 0,Y 156.289,Z 511.437,A -85,B 0,C 180,E1 -23840.363,E2 -23840.363} C_VEL
LIN {X 0,Y 156.093,Z 516.862,A -85,B 0,C 180,E1 -23843.064,E2 -23843.064} C_VEL
LIN {X 0,Y 156.024,Z 521.972,A -85,B 0,C 180,E1 -23846.131,E2 -23846.131} C_VEL
LIN {X 0,Y 156.029,Z 525.562,A -85,B 0,C 180,E1 -23848.715,E2 -23848.715} C_VEL
LIN {X 0,Y 155.904,Z 528.73,A -85,B 0,C 180,E1 -23851.661,E2 -23851.661} C_VEL
LIN {X 0,Y 155.349,Z 529.907,A -85,B 0,C 180,E1 -23853.028,E2 -23853.028} C_VEL
LIN {X 0,Y 153.139,Z 531.622,A -85,B 0,C 180,E1 -23855.776,E2 -23855.776} C_VEL
LIN {X 0,Y 149.621,Z 533.201,A -85,B 0,C 180,E1 -23860.065,E2 -23860.065} C_VEL
LIN {X 0,Y 148.997,Z 533.993,A -85,B 0,C 180,E1 -23862.319,E2 -23862.319} C_VEL
LIN {X 0,Y 149.104,Z 534.125,A -85,B 0,C 180,E1 -23863.074,E2 -23863.074} C_VEL
LIN {X 0,Y 150.174,Z 534.956,A -85,B 0,C 180,E1 -23866.312,E2 -23866.312} C_VEL
LIN {X 0,Y 153.332,Z 534.941,A -85,B 0,C 180,E1 -23871.515,E2 -23871.515} C_VEL
LIN {X 0,Y 155.386,Z 534.412,A -85,B 0,C 180,E1 -23874.024,E2 -23874.024} C_VEL
LIN {X 0,Y 161.184,Z 531.869,A -85,B 0,C 180,E1 -23879.305,E2 -23879.305} C_VEL
LIN {X 0,Y 167.031,Z 528.451,A -85,B 0,C 180,E1 -23883.163,E2 -23883.163} C_VEL
LIN {X 0,Y 172.713,Z 524.53,A -85,B 0,C 180,E1 -23886.161,E2 -23886.161} C_VEL
LIN {X 0,Y 178.913,Z 519.517,A -85,B 0,C 180,E1 -23888.941,E2 -23888.941} C_VEL
LIN {X 0,Y 184.569,Z 514.478,A -85,B 0,C 180,E1 -23891.06,E2 -23891.06} C_VEL
LIN {X 0,Y 190.523,Z 508.452,A -85,B 0,C 180,E1 -23893.034,E2 -23893.034} C_VEL
LIN {X 0,Y 196.794,Z 501.211,A -85,B 0,C 180,E1 -23894.855,E2 -23894.855} C_VEL
LIN {X 0,Y 203.304,Z 492.582,A -85,B 0,C 180,E1 -23896.547,E2 -23896.547} C_VEL
LIN {X 0,Y 208.688,Z 484.404,A -85,B 0,C 180,E1 -23897.807,E2 -23897.807} C_VEL
LIN {X 0,Y 213.623,Z 475.806,A -85,B 0,C 180,E1 -23898.812,E2 -23898.812} C_VEL
LIN {X 0,Y 218.144,Z 466.564,A -85,B 0,C 180,E1 -23899.651,E2 -23899.651} C_VEL
LIN {X 0,Y 222.204,Z 456.571,A -85,B 0,C 180,E1 -23900.348,E2 -23900.348} C_VEL
LIN {X 0,Y 226.658,Z 442.68,A -85,B 0,C 180,E1 -23901.071,E2 -23901.071} C_VEL
LIN {X 0,Y 230.291,Z 425.271,A -85,B 0,C 180,E1 -23901.801,E2 -23901.801} C_VEL
LIN {X 0,Y 229.709,Z 422.722,A -85,B 0,C 180,E1 -23904.181,E2 -23904.181} C_VEL
LIN {X 0,Y 229.379,Z 422.245,A -85,B 0,C 180,E1 -23906.531,E2 -23906.531} C_VEL
LIN {X 0,Y 229.716,Z 422.57,A -85,B 0,C 180,E1 -23909.442,E2 -23909.442} C_VEL
LIN {X 0,Y 230.14,Z 424.591,A -85,B 0,C 180,E1 -23911.392,E2 -23911.392} C_VEL
LIN {X 0,Y 226.389,Z 441.575,A -85,B 0,C 180,E1 -23912.14,E2 -23912.14} C_VEL
LIN {X 0,Y 222.703,Z 452.963,A -85,B 0,C 180,E1 -23912.883,E2 -23912.883} C_VEL
LIN {X 0,Y 219.201,Z 461.63,A -85,B 0,C 180,E1 -23913.587,E2 -23913.587} C_VEL
LIN {X 0,Y 214.776,Z 470.906,A -85,B 0,C 180,E1 -23914.566,E2 -23914.566} C_VEL
LIN {X 0,Y 209.745,Z 479.753,A -85,B 0,C 180,E1 -23915.747,E2 -23915.747} C_VEL
LIN {X 0,Y 204.97,Z 486.966,A -85,B 0,C 180,E1 -23916.965,E2 -23916.965} C_VEL
LIN {X 0,Y 198.623,Z 495.193,A -85,B 0,C 180,E1 -23918.736,E2 -23918.736} C_VEL
LIN {X 0,Y 192.026,Z 502.584,A -85,B 0,C 180,E1 -23920.769,E2 -23920.769} C_VEL
LIN {X 0,Y 184.796,Z 509.356,A -85,B 0,C 180,E1 -23923.35,E2 -23923.35} C_VEL
LIN {X 0,Y 177.797,Z 514.683,A -85,B 0,C 180,E1 -23926.282,E2 -23926.282} C_VEL
LIN {X 0,Y 171.679,Z 518.472,A -85,B 0,C 180,E1 -23929.255,E2 -23929.255} C_VEL
LIN {X 0,Y 167.982,Z 520.298,A -85,B 0,C 180,E1 -23931.362,E2 -23931.362} C_VEL
LIN {X 0,Y 162.198,Z 522.374,A -85,B 0,C 180,E1 -23935.254,E2 -23935.254} C_VEL
LIN {X 0,Y 159.459,Z 522.969,A -85,B 0,C 180,E1 -23937.475,E2 -23937.475} C_VEL
LIN {X 0,Y 156.8,Z 523.04,A -85,B 0,C 180,E1 -23940.001,E2 -23940.001} C_VEL
LIN {X 0,Y 154.447,Z 522.607,A -85,B 0,C 180,E1 -23942.61,E2 -23942.61} C_VEL
LIN {X 0,Y 152.446,Z 521.755,A -85,B 0,C 180,E1 -23945.292,E2 -23945.292} C_VEL
LIN {X 0,Y 150.815,Z 520.427,A -85,B 0,C 180,E1 -23948.038,E2 -23948.038} C_VEL
LIN {X 0,Y 149.062,Z 517.353,A -85,B 0,C 180,E1 -23952.251,E2 -23952.251} C_VEL
LIN {X 0,Y 148.093,Z 513.005,A -85,B 0,C 180,E1 -23956.545,E2 -23956.545} C_VEL
LIN {X 0,Y 147.873,Z 508.292,A -85,B 0,C 180,E1 -23960.157,E2 -23960.157} C_VEL
LIN {X 0,Y 148.017,Z 503.693,A -85,B 0,C 180,E1 -23963.063,E2 -23963.063} C_VEL
LIN {X 0,Y 148.432,Z 497.887,A -85,B 0,C 180,E1 -23966.119,E2 -23966.119} C_VEL
LIN {X 0,Y 148.911,Z 491.48,A -85,B 0,C 180,E1 -23968.933,E2 -23968.933} C_VEL
LIN {X 0,Y 149.706,Z 483.617,A -85,B 0,C 180,E1 -23971.801,E2 -23971.801} C_VEL
LIN {X 0,Y 150.676,Z 474.808,A -85,B 0,C 180,E1 -23974.442,E2 -23974.442} C_VEL
LIN {X 0,Y 151.61,Z 465.767,A -85,B 0,C 180,E1 -23976.645,E2 -23976.645} C_VEL
LIN {X 0,Y 152.712,Z 455.144,A -85,B 0,C 180,E1 -23978.735,E2 -23978.735} C_VEL
LIN {X 0,Y 153.849,Z 442.333,A -85,B 0,C 180,E1 -23980.616,E2 -23980.616} C_VEL
LIN {X 0,Y 154.53,Z 431.041,A -85,B 0,C 180,E1 -23981.804,E2 -23981.804} C_VEL
LIN {X 0,Y 157.396,Z 379.603,A -85,B 0,C 180,E1 -23985.556,E2 -23985.556} C_VEL
LIN {X 0,Y 154.839,Z 348.375,A -85,B 0,C 180,E1 -23988.025,E2 -23988.025} C_VEL
LIN {X 0,Y 154.488,Z 342.239,A -85,B 0,C 180,E1 -23988.509,E2 -23988.509} C_VEL
LIN {X 0,Y 154.264,Z 341.253,A -85,B 0,C 180,E1 -23988.653,E2 -23988.653} C_VEL
LIN {X 0,Y 152.366,Z 331.571,A -85,B 0,C 180,E1 -23993.975,E2 -23993.975} C_VEL
LIN {X 0,Y 150.51,Z 322.798,A -85,B 0,C 180,E1 -23999.091,E2 -23999.091} C_VEL
LIN {X 0,Y 150.252,Z 321.769,A -85,B 0,C 180,E1 -23999.81,E2 -23999.81} C_VEL
LIN {X 0,Y 150.181,Z 321.778,A -85,B 0,C 180,E1 -24005.088,E2 -24005.088} C_VEL
LIN {X 0,Y 150.307,Z 321.762,A -85,B 0,C 180,E1 -24010.891,E2 -24010.891} C_VEL
LIN {X 0,Y 150.419,Z 321.741,A -85,B 0,C 180,E1 -24016.486,E2 -24016.486} C_VEL
LIN {X 0,Y 150.614,Z 321.724,A -85,B 0,C 180,E1 -24019.238,E2 -24019.238} C_VEL
LIN {X 0,Y 150.686,Z 321.713,A -85,B 0,C 180,E1 -24021.952,E2 -24021.952} C_VEL
LIN {X 0,Y 151.2,Z 321.651,A -85,B 0,C 180,E1 -24029.995,E2 -24029.995} C_VEL
LIN {X 0,Y 150.699,Z 321.714,A -85,B 0,C 180,E1 -24038.036,E2 -24038.036} C_VEL
LIN {X 0,Y 150.575,Z 321.724,A -85,B 0,C 180,E1 -24041.424,E2 -24041.424} C_VEL
LIN {X 0,Y 150.321,Z 321.759,A -85,B 0,C 180,E1 -24046.284,E2 -24046.284} C_VEL
LIN {X 0,Y 150.281,Z 321.761,A -85,B 0,C 180,E1 -24050.717,E2 -24050.717} C_VEL
LIN {X 0,Y 150.232,Z 321.772,A -85,B 0,C 180,E1 -24057.269,E2 -24057.269} C_VEL
LIN {X 0,Y 150.199,Z 321.772,A -85,B 0,C 180,E1 -24062.619,E2 -24062.619} C_VEL
LIN {X 0,Y 150.157,Z 321.779,A -85,B 0,C 180,E1 -24067.467,E2 -24067.467} C_VEL
LIN {X 0,Y 150.118,Z 321.782,A -85,B 0,C 180,E1 -24071.489,E2 -24071.489} C_VEL
LIN {X 0,Y 150.11,Z 321.785,A -85,B 0,C 180,E1 -24075.388,E2 -24075.388} C_VEL
LIN {X 0,Y 150.118,Z 321.781,A -85,B 0,C 180,E1 -24079.046,E2 -24079.046} C_VEL
LIN {X 0,Y 150.156,Z 321.782,A -85,B 0,C 180,E1 -24082.703,E2 -24082.703} C_VEL
LIN {X 0,Y 150.192,Z 321.771,A -85,B 0,C 180,E1 -24087.363,E2 -24087.363} C_VEL
LIN {X 0,Y 150.218,Z 321.772,A -85,B 0,C 180,E1 -24092.715,E2 -24092.715} C_VEL
LIN {X 0,Y 150.258,Z 321.767,A -85,B 0,C 180,E1 -24099.272,E2 -24099.272} C_VEL
LIN {X 0,Y 150.286,Z 321.762,A -85,B 0,C 180,E1 -24103.703,E2 -24103.703} C_VEL
LIN {X 0,Y 150.576,Z 321.727,A -85,B 0,C 180,E1 -24109.238,E2 -24109.238} C_VEL
LIN {X 0,Y 150.669,Z 321.715,A -85,B 0,C 180,E1 -24111.954,E2 -24111.954} C_VEL
LIN {X 0,Y 151.18,Z 321.651,A -85,B 0,C 180,E1 -24119.999,E2 -24119.999} C_VEL
LIN {X 0,Y 150.669,Z 321.716,A -85,B 0,C 180,E1 -24128.043,E2 -24128.043} C_VEL
LIN {X 0,Y 150.544,Z 321.727,A -85,B 0,C 180,E1 -24131.428,E2 -24131.428} C_VEL
LIN {X 0,Y 150.314,Z 321.761,A -85,B 0,C 180,E1 -24136.29,E2 -24136.29} C_VEL
LIN {X 0,Y 150.32,Z 321.754,A -85,B 0,C 180,E1 -24140.791,E2 -24140.791} C_VEL
LIN {X 0,Y 150.212,Z 321.771,A -85,B 0,C 180,E1 -24147.281,E2 -24147.281} C_VEL
LIN {X 0,Y 150.182,Z 321.777,A -85,B 0,C 180,E1 -24152.631,E2 -24152.631} C_VEL
LIN {X 0,Y 150.145,Z 321.784,A -85,B 0,C 180,E1 -24157.48,E2 -24157.48} C_VEL
LIN {X 0,Y 150.11,Z 321.789,A -85,B 0,C 180,E1 -24161.502,E2 -24161.502} C_VEL
LIN {X 0,Y 150.18,Z 321.897,A -85,B 0,C 180,E1 -24166.481,E2 -24166.481} C_VEL
LIN {X 0,Y 152.337,Z 331.279,A -85,B 0,C 180,E1 -24171.653,E2 -24171.653} C_VEL
LIN {X 0,Y 154.496,Z 341.433,A -85,B 0,C 180,E1 -24176.925,E2 -24176.925} C_VEL
LIN {X 0,Y 154.934,Z 343.547,A -85,B 0,C 180,E1 -24177.97,E2 -24177.97} C_VEL
LIN {X 0,Y 156.874,Z 351.132,A -85,B 0,C 180,E1 -24178.64,E2 -24178.64} C_VEL
LIN {X 0,Y 158.128,Z 375.869,A -85,B 0,C 180,E1 -24180.414,E2 -24180.414} C_VEL
LIN {X 0,Y 158.644,Z 385.829,A -85,B 0,C 180,E1 -24181.118,E2 -24181.118} C_VEL
LIN {X 0,Y 155.928,Z 441.853,A -85,B 0,C 180,E1 -24184.847,E2 -24184.847} C_VEL
LIN {X 0,Y 155.259,Z 451.652,A -85,B 0,C 180,E1 -24185.791,E2 -24185.791} C_VEL
LIN {X 0,Y 154.309,Z 461.449,A -85,B 0,C 180,E1 -24187.055,E2 -24187.055} C_VEL
LIN {X 0,Y 153.376,Z 470.278,A -85,B 0,C 180,E1 -24188.503,E2 -24188.503} C_VEL
LIN {X 0,Y 152.509,Z 478.456,A -85,B 0,C 180,E1 -24190.14,E2 -24190.14} C_VEL
LIN {X 0,Y 151.398,Z 487.846,A -85,B 0,C 180,E1 -24192.446,E2 -24192.446} C_VEL
LIN {X 0,Y 150.539,Z 495.706,A -85,B 0,C 180,E1 -24194.782,E2 -24194.782} C_VEL
LIN {X 0,Y 149.868,Z 502.372,A -85,B 0,C 180,E1 -24197.136,E2 -24197.136} C_VEL
LIN {X 0,Y 149.362,Z 509.014,A -85,B 0,C 180,E1 -24199.912,E2 -24199.912} C_VEL
LIN {X 0,Y 149.131,Z 516.35,A -85,B 0,C 180,E1 -24203.677,E2 -24203.677} C_VEL
LIN {X 0,Y 149.069,Z 520.132,A -85,B 0,C 180,E1 -24205.951,E2 -24205.951} C_VEL
LIN {X 0,Y 149.13,Z 525.471,A -85,B 0,C 180,E1 -24210.005,E2 -24210.005} C_VEL
LIN {X 0,Y 148.786,Z 528.181,A -85,B 0,C 180,E1 -24212.713,E2 -24212.713} C_VEL
LIN {X 0,Y 148.45,Z 530.862,A -85,B 0,C 180,E1 -24216.19,E2 -24216.19} C_VEL
LIN {X 0,Y 148.63,Z 533.389,A -85,B 0,C 180,E1 -24220.907,E2 -24220.907} C_VEL
LIN {X 0,Y 149.104,Z 534.125,A -85,B 0,C 180,E1 -24223.074,E2 -24223.074} C_VEL
LIN {X 0,Y 149.167,Z 534.711,A -85,B 0,C 180,E1 -24225.333,E2 -24225.333} C_VEL
LIN {X 0,Y 148.061,Z 534.993,A -85,B 0,C 180,E1 -24229.133,E2 -24229.133} C_VEL
LIN {X 0,Y 147.726,Z 534.589,A -85,B 0,C 180,E1 -24232.966,E2 -24232.966} C_VEL
LIN {X 0,Y 148.966,Z 534.102,A -85,B 0,C 180,E1 -24235.185,E2 -24235.185} C_VEL
LIN {X 0,Y 151.485,Z 533.443,A -85,B 0,C 180,E1 -24237.645,E2 -24237.645} C_VEL
LIN {X 0,Y 154.693,Z 532.197,A -85,B 0,C 180,E1 -24240.324,E2 -24240.324} C_VEL
LIN {X 0,Y 161.153,Z 529.044,A -85,B 0,C 180,E1 -24244.539,E2 -24244.539} C_VEL
LIN {X 0,Y 167.095,Z 525.452,A -85,B 0,C 180,E1 -24247.582,E2 -24247.582} C_VEL
LIN {X 0,Y 173.543,Z 520.878,A -85,B 0,C 180,E1 -24250.389,E2 -24250.389} C_VEL
LIN {X 0,Y 180.605,Z 515.087,A -85,B 0,C 180,E1 -24252.922,E2 -24252.922} C_VEL
LIN {X 0,Y 188.071,Z 507.932,A -85,B 0,C 180,E1 -24255.236,E2 -24255.236} C_VEL
LIN {X 0,Y 194.638,Z 500.785,A -85,B 0,C 180,E1 -24256.986,E2 -24256.986} C_VEL
LIN {X 0,Y 200.062,Z 494.082,A -85,B 0,C 180,E1 -24258.287,E2 -24258.287} C_VEL
LIN {X 0,Y 206.388,Z 484.981,A -85,B 0,C 180,E1 -24259.67,E2 -24259.67} C_VEL
LIN {X 0,Y 212.292,Z 475.18,A -85,B 0,C 180,E1 -24260.767,E2 -24260.767} C_VEL
LIN {X 0,Y 217.314,Z 465.272,A -85,B 0,C 180,E1 -24261.605,E2 -24261.605} C_VEL
LIN {X 0,Y 221.994,Z 453.961,A -85,B 0,C 180,E1 -24262.321,E2 -24262.321} C_VEL
LIN {X 0,Y 226.224,Z 440.019,A -85,B 0,C 180,E1 -24262.985,E2 -24262.985} C_VEL
LIN {X 0,Y 228.301,Z 430.603,A -85,B 0,C 180,E1 -24263.388,E2 -24263.388} C_VEL
LIN {X 0,Y 228.144,Z 429.448,A -85,B 0,C 180,E1 -24264.671,E2 -24264.671} C_VEL
LIN {X 0,Y 228.042,Z 429.259,A -85,B 0,C 180,E1 -24268.405,E2 -24268.405} C_VEL
LIN {X 0,Y 228.194,Z 429.757,A -85,B 0,C 180,E1 -24269.579,E2 -24269.579} C_VEL
LIN {X 0,Y 228.163,Z 430.227,A -85,B 0,C 180,E1 -24269.839,E2 -24269.839} C_VEL
LIN {X 0,Y 224.98,Z 443.156,A -85,B 0,C 180,E1 -24270.42,E2 -24270.42} C_VEL
LIN {X 0,Y 220.977,Z 454.88,A -85,B 0,C 180,E1 -24271.165,E2 -24271.165} C_VEL
LIN {X 0,Y 216.755,Z 464.628,A -85,B 0,C 180,E1 -24271.965,E2 -24271.965} C_VEL
LIN {X 0,Y 211.424,Z 474.738,A -85,B 0,C 180,E1 -24273.07,E2 -24273.07} C_VEL
LIN {X 0,Y 204.048,Z 486.019,A -85,B 0,C 180,E1 -24274.721,E2 -24274.721} C_VEL
LIN {X 0,Y 198.897,Z 492.777,A -85,B 0,C 180,E1 -24276.024,E2 -24276.024} C_VEL
LIN {X 0,Y 193.275,Z 499.166,A -85,B 0,C 180,E1 -24277.555,E2 -24277.555} C_VEL
LIN {X 0,Y 187.151,Z 505.137,A -85,B 0,C 180,E1 -24279.359,E2 -24279.359} C_VEL
LIN {X 0,Y 180.019,Z 511.103,A -85,B 0,C 180,E1 -24281.802,E2 -24281.802} C_VEL
LIN {X 0,Y 175.205,Z 514.606,A -85,B 0,C 180,E1 -24283.694,E2 -24283.694} C_VEL
LIN {X 0,Y 168.312,Z 518.633,A -85,B 0,C 180,E1 -24286.724,E2 -24286.724} C_VEL
LIN {X 0,Y 165.004,Z 520.32,A -85,B 0,C 180,E1 -24288.415,E2 -24288.415} C_VEL
LIN {X 0,Y 158.423,Z 522.663,A -85,B 0,C 180,E1 -24292.353,E2 -24292.353} C_VEL
LIN {X 0,Y 155.013,Z 523.399,A -85,B 0,C 180,E1 -24294.799,E2 -24294.799} C_VEL
LIN {X 0,Y 151.969,Z 523.54,A -85,B 0,C 180,E1 -24297.351,E2 -24297.351} C_VEL
LIN {X 0,Y 147.662,Z 522.859,A -85,B 0,C 180,E1 -24301.823,E2 -24301.823} C_VEL
LIN {X 0,Y 144.957,Z 521.295,A -85,B 0,C 180,E1 -24305.566,E2 -24305.566} C_VEL
LIN {X 0,Y 142.73,Z 518.455,A -85,B 0,C 180,E1 -24310.005,E2 -24310.005} C_VEL
LIN {X 0,Y 141.369,Z 514.45,A -85,B 0,C 180,E1 -24314.394,E2 -24314.394} C_VEL
LIN {X 0,Y 140.855,Z 509.489,A -85,B 0,C 180,E1 -24318.556,E2 -24318.556} C_VEL
LIN {X 0,Y 140.982,Z 503.217,A -85,B 0,C 180,E1 -24322.729,E2 -24322.729} C_VEL
LIN {X 0,Y 141.37,Z 497.562,A -85,B 0,C 180,E1 -24325.787,E2 -24325.787} C_VEL
LIN {X 0,Y 141.871,Z 490.873,A -85,B 0,C 180,E1 -24328.802,E2 -24328.802} C_VEL
LIN {X 0,Y 142.596,Z 483.511,A -85,B 0,C 180,E1 -24331.58,E2 -24331.58} C_VEL
LIN {X 0,Y 143.427,Z 475.745,A -85,B 0,C 180,E1 -24334.034,E2 -24334.034} C_VEL
LIN {X 0,Y 144.29,Z 467.541,A -85,B 0,C 180,E1 -24336.2,E2 -24336.2} C_VEL
LIN {X 0,Y 145.225,Z 458.84,A -85,B 0,C 180,E1 -24338.101,E2 -24338.101} C_VEL
LIN {X 0,Y 146.213,Z 448.163,A -85,B 0,C 180,E1 -24339.967,E2 -24339.967} C_VEL
LIN {X 0,Y 147.216,Z 435.28,A -85,B 0,C 180,E1 -24341.65,E2 -24341.65} C_VEL
LIN {X 0,Y 148.349,Z 415.686,A -85,B 0,C 180,E1 -24343.273,E2 -24343.273} C_VEL
LIN {X 0,Y 150.366,Z 379.885,A -85,B 0,C 180,E1 -24345.951,E2 -24345.951} C_VEL
LIN {X 0,Y 147.881,Z 348.829,A -85,B 0,C 180,E1 -24348.523,E2 -24348.523} C_VEL
LIN {X 0,Y 147.464,Z 343.059,A -85,B 0,C 180,E1 -24349.004,E2 -24349.004} C_VEL
LIN {X 0,Y 147.039,Z 341.301,A -85,B 0,C 180,E1 -24349.249,E2 -24349.249} C_VEL
LIN {X 0,Y 145.267,Z 332.147,A -85,B 0,C 180,E1 -24354.507,E2 -24354.507} C_VEL
LIN {X 0,Y 143.367,Z 323.448,A -85,B 0,C 180,E1 -24359.834,E2 -24359.834} C_VEL
LIN {X 0,Y 143.182,Z 322.65,A -85,B 0,C 180,E1 -24360.399,E2 -24360.399} C_VEL
LIN {X 0,Y 143.109,Z 322.66,A -85,B 0,C 180,E1 -24366.863,E2 -24366.863} C_VEL
LIN {X 0,Y 143.253,Z 322.64,A -85,B 0,C 180,E1 -24369.911,E2 -24369.911} C_VEL
LIN {X 0,Y 143.318,Z 322.625,A -85,B 0,C 180,E1 -24375.803,E2 -24375.803} C_VEL
LIN {X 0,Y 143.54,Z 322.603,A -85,B 0,C 180,E1 -24378.701,E2 -24378.701} C_VEL
LIN {X 0,Y 143.612,Z 322.595,A -85,B 0,C 180,E1 -24381.553,E2 -24381.553} C_VEL
LIN {X 0,Y 144.158,Z 322.528,A -85,B 0,C 180,E1 -24389.994,E2 -24389.994} C_VEL
LIN {X 0,Y 143.621,Z 322.595,A -85,B 0,C 180,E1 -24398.435,E2 -24398.435} C_VEL
LIN {X 0,Y 143.501,Z 322.605,A -85,B 0,C 180,E1 -24401.613,E2 -24401.613} C_VEL
LIN {X 0,Y 143.258,Z 322.64,A -85,B 0,C 180,E1 -24407.111,E2 -24407.111} C_VEL
LIN {X 0,Y 143.219,Z 322.638,A -85,B 0,C 180,E1 -24411.189,E2 -24411.189} C_VEL
LIN {X 0,Y 143.176,Z 322.648,A -85,B 0,C 180,E1 -24417.922,E2 -24417.922} C_VEL
LIN {X 0,Y 143.128,Z 322.655,A -85,B 0,C 180,E1 -24423.408,E2 -24423.408} C_VEL
LIN {X 0,Y 143.039,Z 322.661,A -85,B 0,C 180,E1 -24429.685,E2 -24429.685} C_VEL
LIN {X 0,Y 143.018,Z 322.669,A -85,B 0,C 180,E1 -24433.456,E2 -24433.456} C_VEL
LIN {X 0,Y 143.02,Z 322.664,A -85,B 0,C 180,E1 -24437.47,E2 -24437.47} C_VEL
LIN {X 0,Y 143.052,Z 322.664,A -85,B 0,C 180,E1 -24441.802,E2 -24441.802} C_VEL
LIN {X 0,Y 143.159,Z 322.646,A -85,B 0,C 180,E1 -24447.314,E2 -24447.314} C_VEL
LIN {X 0,Y 143.165,Z 322.65,A -85,B 0,C 180,E1 -24452.059,E2 -24452.059} C_VEL
LIN {X 0,Y 143.199,Z 322.645,A -85,B 0,C 180,E1 -24458.796,E2 -24458.796} C_VEL
LIN {X 0,Y 143.226,Z 322.641,A -85,B 0,C 180,E1 -24462.876,E2 -24462.876} C_VEL
LIN {X 0,Y 143.503,Z 322.609,A -85,B 0,C 180,E1 -24468.701,E2 -24468.701} C_VEL
LIN {X 0,Y 143.59,Z 322.596,A -85,B 0,C 180,E1 -24471.555,E2 -24471.555} C_VEL
LIN {X 0,Y 144.14,Z 322.528,A -85,B 0,C 180,E1 -24479.998,E2 -24479.998} C_VEL
LIN {X 0,Y 143.591,Z 322.597,A -85,B 0,C 180,E1 -24488.442,E2 -24488.442} C_VEL
LIN {X 0,Y 143.47,Z 322.608,A -85,B 0,C 180,E1 -24491.617,E2 -24491.617} C_VEL
LIN {X 0,Y 143.253,Z 322.639,A -85,B 0,C 180,E1 -24497.118,E2 -24497.118} C_VEL
LIN {X 0,Y 143.246,Z 322.635,A -85,B 0,C 180,E1 -24501.252,E2 -24501.252} C_VEL
LIN {X 0,Y 143.157,Z 322.65,A -85,B 0,C 180,E1 -24507.934,E2 -24507.934} C_VEL
LIN {X 0,Y 143.113,Z 322.657,A -85,B 0,C 180,E1 -24513.42,E2 -24513.42} C_VEL
LIN {X 0,Y 143.029,Z 322.67,A -85,B 0,C 180,E1 -24519.699,E2 -24519.699} C_VEL
LIN {X 0,Y 143.102,Z 322.77,A -85,B 0,C 180,E1 -24525.813,E2 -24525.813} C_VEL
LIN {X 0,Y 145.175,Z 331.723,A -85,B 0,C 180,E1 -24531.011,E2 -24531.011} C_VEL
LIN {X 0,Y 147.358,Z 341.929,A -85,B 0,C 180,E1 -24536.573,E2 -24536.573} C_VEL
LIN {X 0,Y 147.688,Z 343.493,A -85,B 0,C 180,E1 -24537.394,E2 -24537.394} C_VEL
LIN {X 0,Y 149.936,Z 352.849,A -85,B 0,C 180,E1 -24538.243,E2 -24538.243} C_VEL
LIN {X 0,Y 151.491,Z 381.791,A -85,B 0,C 180,E1 -24540.419,E2 -24540.419} C_VEL
LIN {X 0,Y 151.541,Z 388.132,A -85,B 0,C 180,E1 -24540.869,E2 -24540.869} C_VEL
LIN {X 0,Y 148.858,Z 441.755,A -85,B 0,C 180,E1 -24544.634,E2 -24544.634} C_VEL
LIN {X 0,Y 148.18,Z 451.076,A -85,B 0,C 180,E1 -24545.583,E2 -24545.583} C_VEL
LIN {X 0,Y 147.209,Z 461.438,A -85,B 0,C 180,E1 -24546.999,E2 -24546.999} C_VEL
LIN {X 0,Y 146.27,Z 470.135,A -85,B 0,C 180,E1 -24548.517,E2 -24548.517} C_VEL
LIN {X 0,Y 145.401,Z 478.221,A -85,B 0,C 180,E1 -24550.232,E2 -24550.232} C_VEL
LIN {X 0,Y 144.451,Z 486.341,A -85,B 0,C 180,E1 -24552.305,E2 -24552.305} C_VEL
LIN {X 0,Y 143.478,Z 495.333,A -85,B 0,C 180,E1 -24555.106,E2 -24555.106} C_VEL
LIN {X 0,Y 142.746,Z 502.819,A -85,B 0,C 180,E1 -24557.929,E2 -24557.929} C_VEL
LIN {X 0,Y 142.282,Z 510.581,A -85,B 0,C 180,E1 -24561.485,E2 -24561.485} C_VEL
LIN {X 0,Y 142.163,Z 515.764,A -85,B 0,C 180,E1 -24564.332,E2 -24564.332} C_VEL
LIN {X 0,Y 142.112,Z 520.167,A -85,B 0,C 180,E1 -24567.171,E2 -24567.171} C_VEL
LIN {X 0,Y 142.177,Z 523.803,A -85,B 0,C 180,E1 -24570.006,E2 -24570.006} C_VEL
LIN {X 0,Y 141.874,Z 526.623,A -85,B 0,C 180,E1 -24572.845,E2 -24572.845} C_VEL
LIN {X 0,Y 141.484,Z 529.561,A -85,B 0,C 180,E1 -24576.564,E2 -24576.564} C_VEL
LIN {X 0,Y 141.711,Z 532.31,A -85,B 0,C 180,E1 -24581.447,E2 -24581.447} C_VEL
LIN {X 0,Y 142.375,Z 533.489,A -85,B 0,C 180,E1 -24584.293,E2 -24584.293} C_VEL
LIN {X 0,Y 144.823,Z 534.495,A -85,B 0,C 180,E1 -24589.862,E2 -24589.862} C_VEL
LIN {X 0,Y 146.748,Z 534.565,A -85,B 0,C 180,E1 -24592.531,E2 -24592.531} C_VEL
LIN {X 0,Y 148.966,Z 534.102,A -85,B 0,C 180,E1 -24595.185,E2 -24595.185} C_VEL
LIN {X 0,Y 150.466,Z 533.605,A -85,B 0,C 180,E1 -24597.356,E2 -24597.356} C_VEL
LIN {X 0,Y 153.19,Z 530.803,A -85,B 0,C 180,E1 -24603.922,E2 -24603.922} C_VEL
LIN {X 0,Y 155.276,Z 529.491,A -85,B 0,C 180,E1 -24605.908,E2 -24605.908} C_VEL
LIN {X 0,Y 156.256,Z 529.011,A -85,B 0,C 180,E1 -24606.508,E2 -24606.508} C_VEL
LIN {X 0,Y 163.768,Z 524.958,A -85,B 0,C 180,E1 -24610.071,E2 -24610.071} C_VEL
LIN {X 0,Y 170.655,Z 520.367,A -85,B 0,C 180,E1 -24612.807,E2 -24612.807} C_VEL
LIN {X 0,Y 179.385,Z 513.535,A -85,B 0,C 180,E1 -24615.644,E2 -24615.644} C_VEL
LIN {X 0,Y 185.949,Z 507.572,A -85,B 0,C 180,E1 -24617.477,E2 -24617.477} C_VEL
LIN {X 0,Y 192.779,Z 500.413,A -85,B 0,C 180,E1 -24619.153,E2 -24619.153} C_VEL
LIN {X 0,Y 199.878,Z 491.915,A -85,B 0,C 180,E1 -24620.673,E2 -24620.673} C_VEL
LIN {X 0,Y 204.97,Z 484.922,A -85,B 0,C 180,E1 -24621.658,E2 -24621.658} C_VEL
LIN {X 0,Y 211.106,Z 475.079,A -85,B 0,C 180,E1 -24622.709,E2 -24622.709} C_VEL
LIN {X 0,Y 215.587,Z 466.599,A -85,B 0,C 180,E1 -24623.393,E2 -24623.393} C_VEL
LIN {X 0,Y 220.02,Z 456.624,A -85,B 0,C 180,E1 -24624.019,E2 -24624.019} C_VEL
LIN {X 0,Y 223.768,Z 446.2,A -85,B 0,C 180,E1 -24624.51,E2 -24624.51} C_VEL
LIN {X 0,Y 226.459,Z 436.426,A -85,B 0,C 180,E1 -24624.924,E2 -24624.924} C_VEL
LIN {X 0,Y 226.342,Z 436.094,A -85,B 0,C 180,E1 -24626.021,E2 -24626.021} C_VEL
LIN {X 0,Y 226.381,Z 436.161,A -85,B 0,C 180,E1 -24628.282,E2 -24628.282} C_VEL
LIN {X 0,Y 223.914,Z 445.001,A -85,B 0,C 180,E1 -24628.684,E2 -24628.684} C_VEL
LIN {X 0,Y 219.853,Z 456.138,A -85,B 0,C 180,E1 -24629.372,E2 -24629.372} C_VEL
LIN {X 0,Y 215.355,Z 465.908,A -85,B 0,C 180,E1 -24630.155,E2 -24630.155} C_VEL
LIN {X 0,Y 209.558,Z 476.379,A -85,B 0,C 180,E1 -24631.263,E2 -24631.263} C_VEL
LIN {X 0,Y 202.735,Z 486.316,A -85,B 0,C 180,E1 -24632.658,E2 -24632.658} C_VEL
LIN {X 0,Y 196.855,Z 493.569,A -85,B 0,C 180,E1 -24634.015,E2 -24634.015} C_VEL
LIN {X 0,Y 189.348,Z 501.427,A -85,B 0,C 180,E1 -24635.904,E2 -24635.904} C_VEL
LIN {X 0,Y 183.647,Z 506.6,A -85,B 0,C 180,E1 -24637.501,E2 -24637.501} C_VEL
LIN {X 0,Y 178.188,Z 510.936,A -85,B 0,C 180,E1 -24639.21,E2 -24639.21} C_VEL
LIN {X 0,Y 173.009,Z 514.542,A -85,B 0,C 180,E1 -24641.037,E2 -24641.037} C_VEL
LIN {X 0,Y 165.654,Z 518.739,A -85,B 0,C 180,E1 -24643.994,E2 -24643.994} C_VEL
LIN {X 0,Y 158.384,Z 521.818,A -85,B 0,C 180,E1 -24647.475,E2 -24647.475} C_VEL
LIN {X 0,Y 154.769,Z 523.014,A -85,B 0,C 180,E1 -24649.536,E2 -24649.536} C_VEL
LIN {X 0,Y 148.461,Z 524.038,A -85,B 0,C 180,E1 -24653.782,E2 -24653.782} C_VEL
LIN {X 0,Y 144.465,Z 523.928,A -85,B 0,C 180,E1 -24657.213,E2 -24657.213} C_VEL
LIN {X 0,Y 140.599,Z 522.796,A -85,B 0,C 180,E1 -24661.356,E2 -24661.356} C_VEL
LIN {X 0,Y 136.681,Z 519.502,A -85,B 0,C 180,E1 -24667.387,E2 -24667.387} C_VEL
LIN {X 0,Y 134.898,Z 515.758,A -85,B 0,C 180,E1 -24672.03,E2 -24672.03} C_VEL
LIN {X 0,Y 133.89,Z 509.588,A -85,B 0,C 180,E1 -24677.569,E2 -24677.569} C_VEL
LIN {X 0,Y 133.888,Z 503.894,A -85,B 0,C 180,E1 -24681.56,E2 -24681.56} C_VEL
LIN {X 0,Y 134.208,Z 498.396,A -85,B 0,C 180,E1 -24684.769,E2 -24684.769} C_VEL
LIN {X 0,Y 134.701,Z 491.746,A -85,B 0,C 180,E1 -24688.008,E2 -24688.008} C_VEL
LIN {X 0,Y 135.349,Z 484.76,A -85,B 0,C 180,E1 -24690.85,E2 -24690.85} C_VEL
LIN {X 0,Y 136.237,Z 476.336,A -85,B 0,C 180,E1 -24693.682,E2 -24693.682} C_VEL
LIN {X 0,Y 137.082,Z 468.234,A -85,B 0,C 180,E1 -24695.948,E2 -24695.948} C_VEL
LIN {X 0,Y 138.092,Z 458.842,A -85,B 0,C 180,E1 -24698.106,E2 -24698.106} C_VEL
LIN {X 0,Y 138.992,Z 449.056,A -85,B 0,C 180,E1 -24699.908,E2 -24699.908} C_VEL
LIN {X 0,Y 139.989,Z 438.167,A -85,B 0,C 180,E1 -24701.458,E2 -24701.458} C_VEL
LIN {X 0,Y 140.986,Z 421.875,A -85,B 0,C 180,E1 -24703.025,E2 -24703.025} C_VEL
LIN {X 0,Y 143.281,Z 379.805,A -85,B 0,C 180,E1 -24706.386,E2 -24706.386} C_VEL
LIN {X 0,Y 140.87,Z 347.862,A -85,B 0,C 180,E1 -24709.153,E2 -24709.153} C_VEL
LIN {X 0,Y 140.558,Z 344.495,A -85,B 0,C 180,E1 -24709.455,E2 -24709.455} C_VEL
LIN {X 0,Y 139.841,Z 341.464,A -85,B 0,C 180,E1 -24709.795,E2 -24709.795} C_VEL
LIN {X 0,Y 138.234,Z 333.124,A -85,B 0,C 180,E1 -24714.823,E2 -24714.823} C_VEL
LIN {X 0,Y 136.322,Z 324.5,A -85,B 0,C 180,E1 -24720.345,E2 -24720.345} C_VEL
LIN {X 0,Y 136.14,Z 323.527,A -85,B 0,C 180,E1 -24721.174,E2 -24721.174} C_VEL
LIN {X 0,Y 136.187,Z 323.521,A -85,B 0,C 180,E1 -24728.82,E2 -24728.82} C_VEL
LIN {X 0,Y 136.235,Z 323.509,A -85,B 0,C 180,E1 -24735.048,E2 -24735.048} C_VEL
LIN {X 0,Y 136.432,Z 323.487,A -85,B 0,C 180,E1 -24738.173,E2 -24738.173} C_VEL
LIN {X 0,Y 136.542,Z 323.478,A -85,B 0,C 180,E1 -24741.112,E2 -24741.112} C_VEL
LIN {X 0,Y 137.115,Z 323.405,A -85,B 0,C 180,E1 -24749.994,E2 -24749.994} C_VEL
LIN {X 0,Y 136.548,Z 323.475,A -85,B 0,C 180,E1 -24758.876,E2 -24758.876} C_VEL
LIN {X 0,Y 136.415,Z 323.488,A -85,B 0,C 180,E1 -24761.885,E2 -24761.885} C_VEL
LIN {X 0,Y 136.168,Z 323.522,A -85,B 0,C 180,E1 -24768.032,E2 -24768.032} C_VEL
LIN {X 0,Y 136.144,Z 323.519,A -85,B 0,C 180,E1 -24771.687,E2 -24771.687} C_VEL
LIN {X 0,Y 136.085,Z 323.531,A -85,B 0,C 180,E1 -24778.601,E2 -24778.601} C_VEL
LIN {X 0,Y 136.03,Z 323.539,A -85,B 0,C 180,E1 -24784.622,E2 -24784.622} C_VEL
LIN {X 0,Y 136.011,Z 323.536,A -85,B 0,C 180,E1 -24789.185,E2 -24789.185} C_VEL
LIN {X 0,Y 135.963,Z 323.548,A -85,B 0,C 180,E1 -24793.64,E2 -24793.64} C_VEL
LIN {X 0,Y 135.965,Z 323.543,A -85,B 0,C 180,E1 -24797.779,E2 -24797.779} C_VEL
LIN {X 0,Y 136.001,Z 323.542,A -85,B 0,C 180,E1 -24801.674,E2 -24801.674} C_VEL
LIN {X 0,Y 136.034,Z 323.535,A -85,B 0,C 180,E1 -24805.734,E2 -24805.734} C_VEL
LIN {X 0,Y 136.121,Z 323.528,A -85,B 0,C 180,E1 -24812.309,E2 -24812.309} C_VEL
LIN {X 0,Y 136.163,Z 323.521,A -85,B 0,C 180,E1 -24818.818,E2 -24818.818} C_VEL
LIN {X 0,Y 136.197,Z 323.511,A -85,B 0,C 180,E1 -24825.046,E2 -24825.046} C_VEL
LIN {X 0,Y 136.399,Z 323.494,A -85,B 0,C 180,E1 -24828.175,E2 -24828.175} C_VEL
LIN {X 0,Y 136.517,Z 323.478,A -85,B 0,C 180,E1 -24831.114,E2 -24831.114} C_VEL
LIN {X 0,Y 137.097,Z 323.406,A -85,B 0,C 180,E1 -24839.998,E2 -24839.998} C_VEL
LIN {X 0,Y 136.517,Z 323.479,A -85,B 0,C 180,E1 -24848.883,E2 -24848.883} C_VEL
LIN {X 0,Y 136.386,Z 323.49,A -85,B 0,C 180,E1 -24851.893,E2 -24851.893} C_VEL
LIN {X 0,Y 136.172,Z 323.521,A -85,B 0,C 180,E1 -24858.037,E2 -24858.037} C_VEL
LIN {X 0,Y 136.167,Z 323.517,A -85,B 0,C 180,E1 -24861.746,E2 -24861.746} C_VEL
LIN {X 0,Y 136.067,Z 323.53,A -85,B 0,C 180,E1 -24868.613,E2 -24868.613} C_VEL
LIN {X 0,Y 136.016,Z 323.543,A -85,B 0,C 180,E1 -24874.635,E2 -24874.635} C_VEL
LIN {X 0,Y 136.001,Z 323.546,A -85,B 0,C 180,E1 -24879.199,E2 -24879.199} C_VEL
LIN {X 0,Y 136.04,Z 323.645,A -85,B 0,C 180,E1 -24885.113,E2 -24885.113} C_VEL
LIN {X 0,Y 138.086,Z 332.586,A -85,B 0,C 180,E1 -24890.569,E2 -24890.569} C_VEL
LIN {X 0,Y 139.993,Z 341.379,A -85,B 0,C 180,E1 -24895.629,E2 -24895.629} C_VEL
LIN {X 0,Y 140.424,Z 343.424,A -85,B 0,C 180,E1 -24896.777,E2 -24896.777} C_VEL
LIN {X 0,Y 143.041,Z 354.343,A -85,B 0,C 180,E1 -24897.828,E2 -24897.828} C_VEL
LIN {X 0,Y 144.451,Z 381.569,A -85,B 0,C 180,E1 -24899.976,E2 -24899.976} C_VEL
LIN {X 0,Y 144.536,Z 387.934,A -85,B 0,C 180,E1 -24900.459,E2 -24900.459} C_VEL
LIN {X 0,Y 141.819,Z 440.866,A -85,B 0,C 180,E1 -24904.41,E2 -24904.41} C_VEL
LIN {X 0,Y 141.109,Z 450.715,A -85,B 0,C 180,E1 -24905.454,E2 -24905.454} C_VEL
LIN {X 0,Y 140.136,Z 461.079,A -85,B 0,C 180,E1 -24906.942,E2 -24906.942} C_VEL
LIN {X 0,Y 139.19,Z 469.77,A -85,B 0,C 180,E1 -24908.535,E2 -24908.535} C_VEL
LIN {X 0,Y 138.162,Z 479.284,A -85,B 0,C 180,E1 -24910.701,E2 -24910.701} C_VEL
LIN {X 0,Y 137.183,Z 487.126,A -85,B 0,C 180,E1 -24912.876,E2 -24912.876} C_VEL
LIN {X 0,Y 136.506,Z 493.946,A -85,B 0,C 180,E1 -24915.09,E2 -24915.09} C_VEL
LIN {X 0,Y 135.775,Z 501.589,A -85,B 0,C 180,E1 -24918.058,E2 -24918.058} C_VEL
LIN {X 0,Y 135.355,Z 508.073,A -85,B 0,C 180,E1 -24921.046,E2 -24921.046} C_VEL
LIN {X 0,Y 135.232,Z 514.738,A -85,B 0,C 180,E1 -24924.788,E2 -24924.788} C_VEL
LIN {X 0,Y 135.228,Z 520.104,A -85,B 0,C 180,E1 -24928.517,E2 -24928.517} C_VEL
LIN {X 0,Y 135.255,Z 523.633,A -85,B 0,C 180,E1 -24931.495,E2 -24931.495} C_VEL
LIN {X 0,Y 134.528,Z 528.27,A -85,B 0,C 180,E1 -24936.991,E2 -24936.991} C_VEL
LIN {X 0,Y 134.807,Z 531.209,A -85,B 0,C 180,E1 -24942.041,E2 -24942.041} C_VEL
LIN {X 0,Y 136.625,Z 533.288,A -85,B 0,C 180,E1 -24947.982,E2 -24947.982} C_VEL
LIN {X 0,Y 138.171,Z 533.9,A -85,B 0,C 180,E1 -24950.862,E2 -24950.862} C_VEL
LIN {X 0,Y 142.518,Z 533.825,A -85,B 0,C 180,E1 -24956.351,E2 -24956.351} C_VEL
LIN {X 0,Y 145.212,Z 533.294,A -85,B 0,C 180,E1 -24958.949,E2 -24958.949} C_VEL
LIN {X 0,Y 151.596,Z 531.135,A -85,B 0,C 180,E1 -24963.804,E2 -24963.804} C_VEL
LIN {X 0,Y 156.256,Z 529.011,A -85,B 0,C 180,E1 -24966.508,E2 -24966.508} C_VEL
LIN {X 0,Y 159.004,Z 527.513,A -85,B 0,C 180,E1 -24968.336,E2 -24968.336} C_VEL
LIN {X 0,Y 162.486,Z 524.761,A -85,B 0,C 180,E1 -24971.503,E2 -24971.503} C_VEL
LIN {X 0,Y 166.413,Z 521.346,A -85,B 0,C 180,E1 -24974.422,E2 -24974.422} C_VEL
LIN {X 0,Y 169.736,Z 518.817,A -85,B 0,C 180,E1 -24975.828,E2 -24975.828} C_VEL
LIN {X 0,Y 177.261,Z 513.182,A -85,B 0,C 180,E1 -24978.022,E2 -24978.022} C_VEL
LIN {X 0,Y 184.156,Z 507.298,A -85,B 0,C 180,E1 -24979.753,E2 -24979.753} C_VEL
LIN {X 0,Y 190.837,Z 500.755,A -85,B 0,C 180,E1 -24981.241,E2 -24981.241} C_VEL
LIN {X 0,Y 197.623,Z 493.045,A -85,B 0,C 180,E1 -24982.592,E2 -24982.592} C_VEL
LIN {X 0,Y 204.616,Z 483.756,A -85,B 0,C 180,E1 -24983.818,E2 -24983.818} C_VEL
LIN {X 0,Y 210.057,Z 475.42,A -85,B 0,C 180,E1 -24984.638,E2 -24984.638} C_VEL
LIN {X 0,Y 215.211,Z 466.09,A -85,B 0,C 180,E1 -24985.332,E2 -24985.332} C_VEL
LIN {X 0,Y 219.599,Z 456.498,A -85,B 0,C 180,E1 -24985.892,E2 -24985.892} C_VEL
LIN {X 0,Y 223.259,Z 446.608,A -85,B 0,C 180,E1 -24986.328,E2 -24986.328} C_VEL
LIN {X 0,Y 223.792,Z 444.828,A -85,B 0,C 180,E1 -24986.834,E2 -24986.834} C_VEL
LIN {X 0,Y 219.852,Z 455.55,A -85,B 0,C 180,E1 -24987.458,E2 -24987.458} C_VEL
LIN {X 0,Y 216.132,Z 463.762,A -85,B 0,C 180,E1 -24988.023,E2 -24988.023} C_VEL
LIN {X 0,Y 211.72,Z 471.953,A -85,B 0,C 180,E1 -24988.758,E2 -24988.758} C_VEL
LIN {X 0,Y 206.537,Z 480.092,A -85,B 0,C 180,E1 -24989.673,E2 -24989.673} C_VEL
LIN {X 0,Y 201.078,Z 487.433,A -85,B 0,C 180,E1 -24990.705,E2 -24990.705} C_VEL
LIN {X 0,Y 194.801,Z 494.805,A -85,B 0,C 180,E1 -24992.031,E2 -24992.031} C_VEL
LIN {X 0,Y 187.304,Z 502.26,A -85,B 0,C 180,E1 -24993.781,E2 -24993.781} C_VEL
LIN {X 0,Y 181.146,Z 507.463,A -85,B 0,C 180,E1 -24995.351,E2 -24995.351} C_VEL
LIN {X 0,Y 173.96,Z 512.702,A -85,B 0,C 180,E1 -24997.452,E2 -24997.452} C_VEL
LIN {X 0,Y 168.584,Z 516.067,A -85,B 0,C 180,E1 -24999.248,E2 -24999.248} C_VEL
LIN {X 0,Y 160.878,Z 519.947,A -85,B 0,C 180,E1 -25002.195,E2 -25002.195} C_VEL
LIN {X 0,Y 156.051,Z 521.924,A -85,B 0,C 180,E1 -25004.324,E2 -25004.324} C_VEL
LIN {X 0,Y 150.139,Z 523.614,A -85,B 0,C 180,E1 -25007.378,E2 -25007.378} C_VEL
LIN {X 0,Y 143.505,Z 524.567,A -85,B 0,C 180,E1 -25011.553,E2 -25011.553} C_VEL
LIN {X 0,Y 140.038,Z 524.567,A -85,B 0,C 180,E1 -25014.241,E2 -25014.241} C_VEL
LIN {X 0,Y 136.929,Z 523.963,A -85,B 0,C 180,E1 -25017.06,E2 -25017.06} C_VEL
LIN {X 0,Y 131.929,Z 521.46,A -85,B 0,C 180,E1 -25023.055,E2 -25023.055} C_VEL
LIN {X 0,Y 129.284,Z 518.234,A -85,B 0,C 180,E1 -25027.812,E2 -25027.812} C_VEL
LIN {X 0,Y 128.05,Z 515.441,A -85,B 0,C 180,E1 -25031.137,E2 -25031.137} C_VEL
LIN {X 0,Y 126.99,Z 510.146,A -85,B 0,C 180,E1 -25036.066,E2 -25036.066} C_VEL
LIN {X 0,Y 126.817,Z 504.681,A -85,B 0,C 180,E1 -25040.182,E2 -25040.182} C_VEL
LIN {X 0,Y 127.075,Z 499.141,A -85,B 0,C 180,E1 -25043.641,E2 -25043.641} C_VEL
LIN {X 0,Y 127.58,Z 492.146,A -85,B 0,C 180,E1 -25047.257,E2 -25047.257} C_VEL
LIN {X 0,Y 128.24,Z 484.684,A -85,B 0,C 180,E1 -25050.462,E2 -25050.462} C_VEL
LIN {X 0,Y 129.101,Z 476.427,A -85,B 0,C 180,E1 -25053.409,E2 -25053.409} C_VEL
LIN {X 0,Y 130.068,Z 467.242,A -85,B 0,C 180,E1 -25056.104,E2 -25056.104} C_VEL
LIN {X 0,Y 131.176,Z 456.924,A -85,B 0,C 180,E1 -25058.525,E2 -25058.525} C_VEL
LIN {X 0,Y 132.484,Z 443.372,A -85,B 0,C 180,E1 -25060.904,E2 -25060.904} C_VEL
LIN {X 0,Y 133.272,Z 431.935,A -85,B 0,C 180,E1 -25062.321,E2 -25062.321} C_VEL
LIN {X 0,Y 136.314,Z 380.755,A -85,B 0,C 180,E1 -25066.713,E2 -25066.713} C_VEL
LIN {X 0,Y 134.002,Z 350.027,A -85,B 0,C 180,E1 -25069.528,E2 -25069.528} C_VEL
LIN {X 0,Y 133.541,Z 345.33,A -85,B 0,C 180,E1 -25069.977,E2 -25069.977} C_VEL
LIN {X 0,Y 132.617,Z 341.387,A -85,B 0,C 180,E1 -25070.507,E2 -25070.507} C_VEL
LIN {X 0,Y 130.74,Z 331.917,A -85,B 0,C 180,E1 -25076.561,E2 -25076.561} C_VEL
LIN {X 0,Y 129.088,Z 324.406,A -85,B 0,C 180,E1 -25081.768,E2 -25081.768} C_VEL
LIN {X 0,Y 129.074,Z 324.408,A -85,B 0,C 180,E1 -25087.77,E2 -25087.77} C_VEL
LIN {X 0,Y 129.156,Z 324.394,A -85,B 0,C 180,E1 -25094.207,E2 -25094.207} C_VEL
LIN {X 0,Y 129.35,Z 324.369,A -85,B 0,C 180,E1 -25097.967,E2 -25097.967} C_VEL
LIN {X 0,Y 129.467,Z 324.357,A -85,B 0,C 180,E1 -25100.622,E2 -25100.622} C_VEL
LIN {X 0,Y 130.07,Z 324.283,A -85,B 0,C 180,E1 -25109.994,E2 -25109.994} C_VEL
LIN {X 0,Y 129.471,Z 324.356,A -85,B 0,C 180,E1 -25119.365,E2 -25119.365} C_VEL
LIN {X 0,Y 129.299,Z 324.372,A -85,B 0,C 180,E1 -25122.55,E2 -25122.55} C_VEL
LIN {X 0,Y 129.084,Z 324.404,A -85,B 0,C 180,E1 -25129.058,E2 -25129.058} C_VEL
LIN {X 0,Y 129.041,Z 324.403,A -85,B 0,C 180,E1 -25132.401,E2 -25132.401} C_VEL
LIN {X 0,Y 129.004,Z 324.415,A -85,B 0,C 180,E1 -25135.828,E2 -25135.828} C_VEL
LIN {X 0,Y 129.01,Z 324.41,A -85,B 0,C 180,E1 -25139.349,E2 -25139.349} C_VEL
LIN {X 0,Y 128.946,Z 324.422,A -85,B 0,C 180,E1 -25145.156,E2 -25145.156} C_VEL
LIN {X 0,Y 128.909,Z 324.423,A -85,B 0,C 180,E1 -25150.848,E2 -25150.848} C_VEL
LIN {X 0,Y 128.897,Z 324.427,A -85,B 0,C 180,E1 -25155.124,E2 -25155.124} C_VEL
LIN {X 0,Y 128.916,Z 324.421,A -85,B 0,C 180,E1 -25159.733,E2 -25159.733} C_VEL
LIN {X 0,Y 128.938,Z 324.422,A -85,B 0,C 180,E1 -25164.827,E2 -25164.827} C_VEL
LIN {X 0,Y 128.997,Z 324.415,A -85,B 0,C 180,E1 -25170.635,E2 -25170.635} C_VEL
LIN {X 0,Y 128.991,Z 324.414,A -85,B 0,C 180,E1 -25174.157,E2 -25174.157} C_VEL
LIN {X 0,Y 129.047,Z 324.406,A -85,B 0,C 180,E1 -25177.764,E2 -25177.764} C_VEL
LIN {X 0,Y 129.119,Z 324.394,A -85,B 0,C 180,E1 -25184.206,E2 -25184.206} C_VEL
LIN {X 0,Y 129.317,Z 324.375,A -85,B 0,C 180,E1 -25187.97,E2 -25187.97} C_VEL
LIN {X 0,Y 129.44,Z 324.36,A -85,B 0,C 180,E1 -25190.624,E2 -25190.624} C_VEL
LIN {X 0,Y 130.053,Z 324.283,A -85,B 0,C 180,E1 -25199.998,E2 -25199.998} C_VEL
LIN {X 0,Y 129.44,Z 324.359,A -85,B 0,C 180,E1 -25209.373,E2 -25209.373} C_VEL
LIN {X 0,Y 129.137,Z 324.4,A -85,B 0,C 180,E1 -25215.788,E2 -25215.788} C_VEL
LIN {X 0,Y 129.081,Z 324.402,A -85,B 0,C 180,E1 -25222.273,E2 -25222.273} C_VEL
LIN {X 0,Y 128.997,Z 324.416,A -85,B 0,C 180,E1 -25225.838,E2 -25225.838} C_VEL
LIN {X 0,Y 128.993,Z 324.408,A -85,B 0,C 180,E1 -25229.362,E2 -25229.362} C_VEL
LIN {X 0,Y 128.931,Z 324.424,A -85,B 0,C 180,E1 -25235.17,E2 -25235.17} C_VEL
LIN {X 0,Y 128.9,Z 324.431,A -85,B 0,C 180,E1 -25240.862,E2 -25240.862} C_VEL
LIN {X 0,Y 128.956,Z 324.456,A -85,B 0,C 180,E1 -25244.335,E2 -25244.335} C_VEL
LIN {X 0,Y 131.087,Z 333.772,A -85,B 0,C 180,E1 -25250.339,E2 -25250.339} C_VEL
LIN {X 0,Y 133.191,Z 343.383,A -85,B 0,C 180,E1 -25256.128,E2 -25256.128} C_VEL
LIN {X 0,Y 136.098,Z 355.35,A -85,B 0,C 180,E1 -25257.372,E2 -25257.372} C_VEL
LIN {X 0,Y 137.34,Z 380.847,A -85,B 0,C 180,E1 -25259.5,E2 -25259.5} C_VEL
LIN {X 0,Y 137.549,Z 387.234,A -85,B 0,C 180,E1 -25260.018,E2 -25260.018} C_VEL
LIN {X 0,Y 134.753,Z 440.489,A -85,B 0,C 180,E1 -25264.214,E2 -25264.214} C_VEL
LIN {X 0,Y 134.042,Z 450.347,A -85,B 0,C 180,E1 -25265.313,E2 -25265.313} C_VEL
LIN {X 0,Y 133.043,Z 460.687,A -85,B 0,C 180,E1 -25266.875,E2 -25266.875} C_VEL
LIN {X 0,Y 132.106,Z 469.397,A -85,B 0,C 180,E1 -25268.555,E2 -25268.555} C_VEL
LIN {X 0,Y 131.071,Z 478.9,A -85,B 0,C 180,E1 -25270.836,E2 -25270.836} C_VEL
LIN {X 0,Y 130.004,Z 487.882,A -85,B 0,C 180,E1 -25273.52,E2 -25273.52} C_VEL
LIN {X 0,Y 129.311,Z 494.434,A -85,B 0,C 180,E1 -25275.851,E2 -25275.851} C_VEL
LIN {X 0,Y 128.677,Z 501.883,A -85,B 0,C 180,E1 -25278.989,E2 -25278.989} C_VEL
LIN {X 0,Y 128.384,Z 508.205,A -85,B 0,C 180,E1 -25282.141,E2 -25282.141} C_VEL
LIN {X 0,Y 128.386,Z 514.743,A -85,B 0,C 180,E1 -25286.083,E2 -25286.083} C_VEL
LIN {X 0,Y 128.367,Z 519.966,A -85,B 0,C 180,E1 -25290.006,E2 -25290.006} C_VEL
LIN {X 0,Y 128.395,Z 521.722,A -85,B 0,C 180,E1 -25291.574,E2 -25291.574} C_VEL
LIN {X 0,Y 127.88,Z 524.679,A -85,B 0,C 180,E1 -25294.735,E2 -25294.735} C_VEL
LIN {X 0,Y 127.629,Z 528.136,A -85,B 0,C 180,E1 -25299.514,E2 -25299.514} C_VEL
LIN {X 0,Y 127.951,Z 529.967,A -85,B 0,C 180,E1 -25302.697,E2 -25302.697} C_VEL
LIN {X 0,Y 129.906,Z 532.436,A -85,B 0,C 180,E1 -25308.946,E2 -25308.946} C_VEL
LIN {X 0,Y 133.748,Z 533.409,A -85,B 0,C 180,E1 -25314.862,E2 -25314.862} C_VEL
LIN {X 0,Y 136.188,Z 533.456,A -85,B 0,C 180,E1 -25317.678,E2 -25317.678} C_VEL
LIN {X 0,Y 142.212,Z 532.359,A -85,B 0,C 180,E1 -25322.933,E2 -25322.933} C_VEL
LIN {X 0,Y 149.703,Z 529.785,A -85,B 0,C 180,E1 -25327.614,E2 -25327.614} C_VEL
LIN {X 0,Y 153.875,Z 528.029,A -85,B 0,C 180,E1 -25329.751,E2 -25329.751} C_VEL
LIN {X 0,Y 163.102,Z 523.06,A -85,B 0,C 180,E1 -25333.587,E2 -25333.587} C_VEL
LIN {X 0,Y 169.736,Z 518.817,A -85,B 0,C 180,E1 -25335.828,E2 -25335.828} C_VEL
LIN {X 0,Y 173.197,Z 516.169,A -85,B 0,C 180,E1 -25337.16,E2 -25337.16} C_VEL
LIN {X 0,Y 182.337,Z 507.635,A -85,B 0,C 180,E1 -25341.671,E2 -25341.671} C_VEL
LIN {X 0,Y 185.181,Z 504.831,A -85,B 0,C 180,E1 -25342.576,E2 -25342.576} C_VEL
LIN {X 0,Y 186.444,Z 503.636,A -85,B 0,C 180,E1 -25342.865,E2 -25342.865} C_VEL
LIN {X 0,Y 195.591,Z 494.335,A -85,B 0,C 180,E1 -25344.539,E2 -25344.539} C_VEL
LIN {X 0,Y 203.831,Z 483.979,A -85,B 0,C 180,E1 -25345.842,E2 -25345.842} C_VEL
LIN {X 0,Y 210.21,Z 474.374,A -85,B 0,C 180,E1 -25346.701,E2 -25346.701} C_VEL
LIN {X 0,Y 209.148,Z 476.005,A -85,B 0,C 180,E1 -25347.146,E2 -25347.146} C_VEL
LIN {X 0,Y 201.43,Z 486.765,A -85,B 0,C 180,E1 -25348.443,E2 -25348.443} C_VEL
LIN {X 0,Y 194.817,Z 494.338,A -85,B 0,C 180,E1 -25349.667,E2 -25349.667} C_VEL
LIN {X 0,Y 186.907,Z 501.934,A -85,B 0,C 180,E1 -25351.305,E2 -25351.305} C_VEL
LIN {X 0,Y 180.527,Z 507.28,A -85,B 0,C 180,E1 -25352.78,E2 -25352.78} C_VEL
LIN {X 0,Y 175.935,Z 510.712,A -85,B 0,C 180,E1 -25353.935,E2 -25353.935} C_VEL
LIN {X 0,Y 167.153,Z 516.124,A -85,B 0,C 180,E1 -25356.457,E2 -25356.457} C_VEL
LIN {X 0,Y 158.929,Z 520.144,A -85,B 0,C 180,E1 -25359.284,E2 -25359.284} C_VEL
LIN {X 0,Y 153.745,Z 522.211,A -85,B 0,C 180,E1 -25361.34,E2 -25361.34} C_VEL
LIN {X 0,Y 145.313,Z 524.386,A -85,B 0,C 180,E1 -25365.306,E2 -25365.306} C_VEL
LIN {X 0,Y 139.964,Z 525.094,A -85,B 0,C 180,E1 -25368.415,E2 -25368.415} C_VEL
LIN {X 0,Y 134.846,Z 525.025,A -85,B 0,C 180,E1 -25371.997,E2 -25371.997} C_VEL
LIN {X 0,Y 129.416,Z 523.694,A -85,B 0,C 180,E1 -25376.889,E2 -25376.889} C_VEL
LIN {X 0,Y 126.507,Z 522.221,A -85,B 0,C 180,E1 -25380.242,E2 -25380.242} C_VEL
LIN {X 0,Y 123.446,Z 519.323,A -85,B 0,C 180,E1 -25384.901,E2 -25384.901} C_VEL
LIN {X 0,Y 121.28,Z 515.123,A -85,B 0,C 180,E1 -25390.013,E2 -25390.013} C_VEL
LIN {X 0,Y 120.201,Z 510.619,A -85,B 0,C 180,E1 -25394.39,E2 -25394.39} C_VEL
LIN {X 0,Y 119.866,Z 505.345,A -85,B 0,C 180,E1 -25398.643,E2 -25398.643} C_VEL
LIN {X 0,Y 119.973,Z 499.817,A -85,B 0,C 180,E1 -25402.383,E2 -25402.383} C_VEL
LIN {X 0,Y 120.375,Z 493.456,A -85,B 0,C 180,E1 -25405.971,E2 -25405.971} C_VEL
LIN {X 0,Y 121.177,Z 484.282,A -85,B 0,C 180,E1 -25410.139,E2 -25410.139} C_VEL
LIN {X 0,Y 122.016,Z 476.131,A -85,B 0,C 180,E1 -25413.177,E2 -25413.177} C_VEL
LIN {X 0,Y 122.955,Z 467.232,A -85,B 0,C 180,E1 -25415.913,E2 -25415.913} C_VEL
LIN {X 0,Y 124.093,Z 456.673,A -85,B 0,C 180,E1 -25418.537,E2 -25418.537} C_VEL
LIN {X 0,Y 125.317,Z 443.663,A -85,B 0,C 180,E1 -25420.956,E2 -25420.956} C_VEL
LIN {X 0,Y 126.129,Z 432.56,A -85,B 0,C 180,E1 -25422.436,E2 -25422.436} C_VEL
LIN {X 0,Y 128.762,Z 389.609,A -85,B 0,C 180,E1 -25426.393,E2 -25426.393} C_VEL
